LIN {X 0,Y 256.462,Z 255.037,A -85,B 0,C 180,E1 -18622.127,E2 -18622.127} C_VEL
LIN {X 0,Y 256.466,Z 255.038,A -85,B 0,C 180,E1 -18626.861,E2 -18626.861} C_VEL
LIN {X 0,Y 256.7,Z 255.004,A -85,B 0,C 180,E1 -18630.003,E2 -18630.003} C_VEL
LIN {X 0,Y 256.467,Z 255.035,A -85,B 0,C 180,E1 -18633.144,E2 -18633.144} C_VEL
LIN {X 0,Y 256.467,Z 255.036,A -85,B 0,C 180,E1 -18637.878,E2 -18637.878} C_VEL
LIN {X 0,Y 256.243,Z 255.057,A -85,B 0,C 180,E1 -18641.071,E2 -18641.071} C_VEL
LIN {X 0,Y 256.205,Z 255.066,A -85,B 0,C 180,E1 -18645.924,E2 -18645.924} C_VEL
LIN {X 0,Y 256.125,Z 255.068,A -85,B 0,C 180,E1 -18649.227,E2 -18649.227} C_VEL
LIN {X 0,Y 256.028,Z 255.091,A -85,B 0,C 180,E1 -18652.603,E2 -18652.603} C_VEL
LIN {X 0,Y 256.077,Z 255.079,A -85,B 0,C 180,E1 -18656.05,E2 -18656.05} C_VEL
LIN {X 0,Y 256.055,Z 255.069,A -85,B 0,C 180,E1 -18659.61,E2 -18659.61} C_VEL
LIN {X 0,Y 256.039,Z 255.087,A -85,B 0,C 180,E1 -18663.3,E2 -18663.3} C_VEL
LIN {X 0,Y 256.09,Z 255.081,A -85,B 0,C 180,E1 -18667.286,E2 -18667.286} C_VEL
LIN {X 0,Y 256.066,Z 255.085,A -85,B 0,C 180,E1 -18671.204,E2 -18671.204} C_VEL
LIN {X 0,Y 256.081,Z 255.085,A -85,B 0,C 180,E1 -18674.494,E2 -18674.494} C_VEL
LIN {X 0,Y 256.128,Z 255.08,A -85,B 0,C 180,E1 -18678.828,E2 -18678.828} C_VEL
LIN {X 0,Y 256.128,Z 255.078,A -85,B 0,C 180,E1 -18682.883,E2 -18682.883} C_VEL
LIN {X 0,Y 256.062,Z 255.083,A -85,B 0,C 180,E1 -18686.721,E2 -18686.721} C_VEL
LIN {X 0,Y 256.107,Z 255.081,A -85,B 0,C 180,E1 -18691.422,E2 -18691.422} C_VEL
LIN {X 0,Y 256.127,Z 255.076,A -85,B 0,C 180,E1 -18695.708,E2 -18695.708} C_VEL
LIN {X 0,Y 256.115,Z 255.082,A -85,B 0,C 180,E1 -18699.113,E2 -18699.113} C_VEL
LIN {X 0,Y 256.224,Z 255.06,A -85,B 0,C 180,E1 -18704.092,E2 -18704.092} C_VEL
LIN {X 0,Y 256.285,Z 255.059,A -85,B 0,C 180,E1 -18707.339,E2 -18707.339} C_VEL
LIN {X 0,Y 256.435,Z 255.037,A -85,B 0,C 180,E1 -18710.634,E2 -18710.634} C_VEL
LIN {X 0,Y 256.459,Z 255.032,A -85,B 0,C 180,E1 -18713.718,E2 -18713.718} C_VEL
LIN {X 0,Y 256.705,Z 255.007,A -85,B 0,C 180,E1 -18718.442,E2 -18718.442} C_VEL
LIN {X 0,Y 256.708,Z 255.001,A -85,B 0,C 180,E1 -18721.579,E2 -18721.579} C_VEL
LIN {X 0,Y 256.314,Z 255.029,A -85,B 0,C 180,E1 -18724.838,E2 -18724.838} C_VEL
LIN {X 0,Y 255.699,Z 255.11,A -85,B 0,C 180,E1 -18726.152,E2 -18726.152} C_VEL
LIN {X 0,Y 252.868,Z 255.475,A -85,B 0,C 180,E1 -18728.293,E2 -18728.293} C_VEL
LIN {X 0,Y 250.409,Z 255.789,A -85,B 0,C 180,E1 -18730.035,E2 -18730.035} C_VEL
LIN {X 0,Y 249.32,Z 255.926,A -85,B 0,C 180,E1 -18731.387,E2 -18731.387} C_VEL
LIN {X 0,Y 249.215,Z 255.937,A -85,B 0,C 180,E1 -18731.846,E2 -18731.846} C_VEL
LIN {X 0,Y 249.193,Z 255.935,A -85,B 0,C 180,E1 -18736.476,E2 -18736.476} C_VEL
LIN {X 0,Y 249.068,Z 255.955,A -85,B 0,C 180,E1 -18741.53,E2 -18741.53} C_VEL
LIN {X 0,Y 249.107,Z 255.952,A -85,B 0,C 180,E1 -18745.466,E2 -18745.466} C_VEL
LIN {X 0,Y 249.053,Z 255.95,A -85,B 0,C 180,E1 -18748.976,E2 -18748.976} C_VEL
LIN {X 0,Y 249.052,Z 255.96,A -85,B 0,C 180,E1 -18752.433,E2 -18752.433} C_VEL
LIN {X 0,Y 249.038,Z 255.951,A -85,B 0,C 180,E1 -18756.354,E2 -18756.354} C_VEL
LIN {X 0,Y 249.003,Z 255.965,A -85,B 0,C 180,E1 -18760.489,E2 -18760.489} C_VEL
LIN {X 0,Y 248.981,Z 255.971,A -85,B 0,C 180,E1 -18765.113,E2 -18765.113} C_VEL
LIN {X 0,Y 249.001,Z 255.968,A -85,B 0,C 180,E1 -18769.659,E2 -18769.659} C_VEL
LIN {X 0,Y 249.041,Z 255.964,A -85,B 0,C 180,E1 -18773.654,E2 -18773.654} C_VEL
LIN {X 0,Y 249.103,Z 256.071,A -85,B 0,C 180,E1 -18775.646,E2 -18775.646} C_VEL
LIN {X 0,Y 250.915,Z 264.838,A -85,B 0,C 180,E1 -18779.255,E2 -18779.255} C_VEL
LIN {X 0,Y 251.505,Z 267.617,A -85,B 0,C 180,E1 -18780.284,E2 -18780.284} C_VEL
LIN {X 0,Y 258.173,Z 286.572,A -85,B 0,C 180,E1 -18781.623,E2 -18781.623} C_VEL
LIN {X 0,Y 261.815,Z 312.545,A -85,B 0,C 180,E1 -18782.819,E2 -18782.819} C_VEL
LIN {X 0,Y 259.494,Z 375.05,A -85,B 0,C 180,E1 -18784.748,E2 -18784.748} C_VEL
LIN {X 0,Y 258.565,Z 388.595,A -85,B 0,C 180,E1 -18785.456,E2 -18785.456} C_VEL
LIN {X 0,Y 257.311,Z 401.593,A -85,B 0,C 180,E1 -18786.453,E2 -18786.453} C_VEL
LIN {X 0,Y 255.62,Z 414.247,A -85,B 0,C 180,E1 -18787.785,E2 -18787.785} C_VEL
LIN {X 0,Y 253.952,Z 425.589,A -85,B 0,C 180,E1 -18789.336,E2 -18789.336} C_VEL
LIN {X 0,Y 252.459,Z 435.754,A -85,B 0,C 180,E1 -18791.095,E2 -18791.095} C_VEL
LIN {X 0,Y 251.161,Z 444.272,A -85,B 0,C 180,E1 -18792.911,E2 -18792.911} C_VEL
LIN {X 0,Y 249.841,Z 452.028,A -85,B 0,C 180,E1 -18794.915,E2 -18794.915} C_VEL
LIN {X 0,Y 248.545,Z 459.611,A -85,B 0,C 180,E1 -18797.339,E2 -18797.339} C_VEL
LIN {X 0,Y 247.864,Z 464.765,A -85,B 0,C 180,E1 -18799.377,E2 -18799.377} C_VEL
LIN {X 0,Y 247.297,Z 469.736,A -85,B 0,C 180,E1 -18801.828,E2 -18801.828} C_VEL
LIN {X 0,Y 246.944,Z 473.528,A -85,B 0,C 180,E1 -18804.281,E2 -18804.281} C_VEL
LIN {X 0,Y 246.853,Z 476.257,A -85,B 0,C 180,E1 -18806.733,E2 -18806.733} C_VEL
LIN {X 0,Y 246.876,Z 477.532,A -85,B 0,C 180,E1 -18808.366,E2 -18808.366} C_VEL
LIN {X 0,Y 246.908,Z 478.388,A -85,B 0,C 180,E1 -18809.997,E2 -18809.997} C_VEL
LIN {X 0,Y 246.873,Z 478.79,A -85,B 0,C 180,E1 -18811.629,E2 -18811.629} C_VEL
LIN {X 0,Y 246.91,Z 478.408,A -85,B 0,C 180,E1 -18814.896,E2 -18814.896} C_VEL
LIN {X 0,Y 247.108,Z 477.628,A -85,B 0,C 180,E1 -18816.529,E2 -18816.529} C_VEL
LIN {X 0,Y 247.419,Z 476.405,A -85,B 0,C 180,E1 -18818.162,E2 -18818.162} C_VEL
LIN {X 0,Y 248.163,Z 473.816,A -85,B 0,C 180,E1 -18820.605,E2 -18820.605} C_VEL
LIN {X 0,Y 249.262,Z 470.223,A -85,B 0,C 180,E1 -18823.033,E2 -18823.033} C_VEL
LIN {X 0,Y 250.734,Z 465.534,A -85,B 0,C 180,E1 -18825.44,E2 -18825.44} C_VEL
LIN {X 0,Y 253.142,Z 458.477,A -85,B 0,C 180,E1 -18828.197,E2 -18828.197} C_VEL
LIN {X 0,Y 255.47,Z 451.067,A -85,B 0,C 180,E1 -18830.482,E2 -18830.482} C_VEL
LIN {X 0,Y 257.729,Z 443.236,A -85,B 0,C 180,E1 -18832.44,E2 -18832.44} C_VEL
LIN {X 0,Y 260.587,Z 432.866,A -85,B 0,C 180,E1 -18834.495,E2 -18834.495} C_VEL
LIN {X 0,Y 263.36,Z 422.361,A -85,B 0,C 180,E1 -18836.121,E2 -18836.121} C_VEL
LIN {X 0,Y 265.495,Z 412.353,A -85,B 0,C 180,E1 -18837.38,E2 -18837.38} C_VEL
LIN {X 0,Y 267.92,Z 399.574,A -85,B 0,C 180,E1 -18838.599,E2 -18838.599} C_VEL
LIN {X 0,Y 269.848,Z 386.608,A -85,B 0,C 180,E1 -18839.495,E2 -18839.495} C_VEL
LIN {X 0,Y 271.208,Z 373.712,A -85,B 0,C 180,E1 -18840.096,E2 -18840.096} C_VEL
LIN {X 0,Y 274.368,Z 315.731,A -85,B 0,C 180,E1 -18841.897,E2 -18841.897} C_VEL
LIN {X 0,Y 272.677,Z 304.843,A -85,B 0,C 180,E1 -18842.649,E2 -18842.649} C_VEL
LIN {X 0,Y 268.046,Z 294.247,A -85,B 0,C 180,E1 -18843.981,E2 -18843.981} C_VEL
LIN {X 0,Y 262.592,Z 283.414,A -85,B 0,C 180,E1 -18845.624,E2 -18845.624} C_VEL
LIN {X 0,Y 257.789,Z 275.094,A -85,B 0,C 180,E1 -18847.131,E2 -18847.131} C_VEL
LIN {X 0,Y 254.919,Z 270.398,A -85,B 0,C 180,E1 -18848.092,E2 -18848.092} C_VEL
LIN {X 0,Y 252.035,Z 265.64,A -85,B 0,C 180,E1 -18849.18,E2 -18849.18} C_VEL
LIN {X 0,Y 249.945,Z 259.149,A -85,B 0,C 180,E1 -18853.012,E2 -18853.012} C_VEL
LIN {X 0,Y 249.001,Z 256,A -85,B 0,C 180,E1 -18855.252,E2 -18855.252} C_VEL
LIN {X 0,Y 248.992,Z 255.969,A -85,B 0,C 180,E1 -18859.644,E2 -18859.644} C_VEL
LIN {X 0,Y 249.019,Z 255.958,A -85,B 0,C 180,E1 -18863.643,E2 -18863.643} C_VEL
LIN {X 0,Y 249.037,Z 255.96,A -85,B 0,C 180,E1 -18867.84,E2 -18867.84} C_VEL
LIN {X 0,Y 249.043,Z 255.96,A -85,B 0,C 180,E1 -18871.322,E2 -18871.322} C_VEL
LIN {X 0,Y 249.103,Z 255.952,A -85,B 0,C 180,E1 -18874.954,E2 -18874.954} C_VEL
LIN {X 0,Y 249.053,Z 255.96,A -85,B 0,C 180,E1 -18878.617,E2 -18878.617} C_VEL
LIN {X 0,Y 249.155,Z 255.943,A -85,B 0,C 180,E1 -18883.606,E2 -18883.606} C_VEL
LIN {X 0,Y 249.212,Z 255.935,A -85,B 0,C 180,E1 -18888.605,E2 -18888.605} C_VEL
LIN {X 0,Y 249.406,Z 255.912,A -85,B 0,C 180,E1 -18891.89,E2 -18891.89} C_VEL
LIN {X 0,Y 249.255,Z 255.932,A -85,B 0,C 180,E1 -18895.137,E2 -18895.137} C_VEL
LIN {X 0,Y 249.648,Z 255.887,A -85,B 0,C 180,E1 -18898.376,E2 -18898.376} C_VEL
LIN {X 0,Y 249.657,Z 255.886,A -85,B 0,C 180,E1 -18901.602,E2 -18901.602} C_VEL
LIN {X 0,Y 249.451,Z 256.029,A -85,B 0,C 180,E1 -18903.219,E2 -18903.219} C_VEL
LIN {X 0,Y 251.162,Z 261.37,A -85,B 0,C 180,E1 -18906.617,E2 -18906.617} C_VEL
LIN {X 0,Y 254.131,Z 265.956,A -85,B 0,C 180,E1 -18907.737,E2 -18907.737} C_VEL
LIN {X 0,Y 258.847,Z 273.575,A -85,B 0,C 180,E1 -18909.315,E2 -18909.315} C_VEL
LIN {X 0,Y 265.164,Z 284.458,A -85,B 0,C 180,E1 -18911.246,E2 -18911.246} C_VEL
LIN {X 0,Y 270.999,Z 296.328,A -85,B 0,C 180,E1 -18912.943,E2 -18912.943} C_VEL
LIN {X 0,Y 274.837,Z 305.474,A -85,B 0,C 180,E1 -18914.031,E2 -18914.031} C_VEL
LIN {X 0,Y 271.212,Z 369.796,A -85,B 0,C 180,E1 -18916.039,E2 -18916.039} C_VEL
LIN {X 0,Y 269.677,Z 383.672,A -85,B 0,C 180,E1 -18916.745,E2 -18916.745} C_VEL
LIN {X 0,Y 268.02,Z 395.502,A -85,B 0,C 180,E1 -18917.638,E2 -18917.638} C_VEL
LIN {X 0,Y 265.705,Z 407.921,A -85,B 0,C 180,E1 -18918.894,E2 -18918.894} C_VEL
LIN {X 0,Y 263.365,Z 418.563,A -85,B 0,C 180,E1 -18920.286,E2 -18920.286} C_VEL
LIN {X 0,Y 260.75,Z 428.824,A -85,B 0,C 180,E1 -18921.968,E2 -18921.968} C_VEL
LIN {X 0,Y 258.22,Z 437.668,A -85,B 0,C 180,E1 -18923.782,E2 -18923.782} C_VEL
LIN {X 0,Y 255.435,Z 446.676,A -85,B 0,C 180,E1 -18926.105,E2 -18926.105} C_VEL
LIN {X 0,Y 252.942,Z 454.285,A -85,B 0,C 180,E1 -18928.599,E2 -18928.599} C_VEL
LIN {X 0,Y 250.854,Z 460.406,A -85,B 0,C 180,E1 -18931.204,E2 -18931.204} C_VEL
LIN {X 0,Y 249.511,Z 464.384,A -85,B 0,C 180,E1 -18933.369,E2 -18933.369} C_VEL
LIN {X 0,Y 248.057,Z 468.539,A -85,B 0,C 180,E1 -18936.495,E2 -18936.495} C_VEL
LIN {X 0,Y 247.091,Z 471.202,A -85,B 0,C 180,E1 -18939.834,E2 -18939.834} C_VEL
LIN {X 0,Y 246.59,Z 472.14,A -85,B 0,C 180,E1 -18943.14,E2 -18943.14} C_VEL
LIN {X 0,Y 246.467,Z 471.807,A -85,B 0,C 180,E1 -18945.45,E2 -18945.45} C_VEL
LIN {X 0,Y 246.455,Z 470.618,A -85,B 0,C 180,E1 -18947.832,E2 -18947.832} C_VEL
LIN {X 0,Y 246.642,Z 468.47,A -85,B 0,C 180,E1 -18950.275,E2 -18950.275} C_VEL
LIN {X 0,Y 247.058,Z 465.231,A -85,B 0,C 180,E1 -18952.775,E2 -18952.775} C_VEL
LIN {X 0,Y 247.691,Z 460.527,A -85,B 0,C 180,E1 -18955.429,E2 -18955.429} C_VEL
LIN {X 0,Y 248.603,Z 454.629,A -85,B 0,C 180,E1 -18957.979,E2 -18957.979} C_VEL
LIN {X 0,Y 249.514,Z 448.37,A -85,B 0,C 180,E1 -18960.142,E2 -18960.142} C_VEL
LIN {X 0,Y 250.916,Z 440.001,A -85,B 0,C 180,E1 -18962.478,E2 -18962.478} C_VEL
LIN {X 0,Y 252.491,Z 430.143,A -85,B 0,C 180,E1 -18964.665,E2 -18964.665} C_VEL
LIN {X 0,Y 254.061,Z 420.365,A -85,B 0,C 180,E1 -18966.41,E2 -18966.41} C_VEL
LIN {X 0,Y 255.514,Z 410.22,A -85,B 0,C 180,E1 -18967.875,E2 -18967.875} C_VEL
LIN {X 0,Y 257.062,Z 397.642,A -85,B 0,C 180,E1 -18969.289,E2 -18969.289} C_VEL
LIN {X 0,Y 258.251,Z 385.45,A -85,B 0,C 180,E1 -18970.323,E2 -18970.323} C_VEL
LIN {X 0,Y 259.236,Z 373.09,A -85,B 0,C 180,E1 -18971.065,E2 -18971.065} C_VEL
LIN {X 0,Y 260.034,Z 356.998,A -85,B 0,C 180,E1 -18971.647,E2 -18971.647} C_VEL
LIN {X 0,Y 262.026,Z 299.434,A -85,B 0,C 180,E1 -18973.409,E2 -18973.409} C_VEL
LIN {X 0,Y 260.034,Z 288.531,A -85,B 0,C 180,E1 -18973.952,E2 -18973.952} C_VEL
LIN {X 0,Y 250.328,Z 261.517,A -85,B 0,C 180,E1 -18975.834,E2 -18975.834} C_VEL
LIN {X 0,Y 250.056,Z 260.316,A -85,B 0,C 180,E1 -18976.182,E2 -18976.182} C_VEL
LIN {X 0,Y 249.212,Z 256.009,A -85,B 0,C 180,E1 -18978.102,E2 -18978.102} C_VEL
LIN {X 0,Y 249.4,Z 255.917,A -85,B 0,C 180,E1 -18981.903,E2 -18981.903} C_VEL
LIN {X 0,Y 249.401,Z 255.917,A -85,B 0,C 180,E1 -18986.772,E2 -18986.772} C_VEL
LIN {X 0,Y 249.663,Z 255.88,A -85,B 0,C 180,E1 -18990.003,E2 -18990.003} C_VEL
LIN {X 0,Y 249.401,Z 255.914,A -85,B 0,C 180,E1 -18993.234,E2 -18993.234} C_VEL
LIN {X 0,Y 249.408,Z 255.915,A -85,B 0,C 180,E1 -18998.102,E2 -18998.102} C_VEL
LIN {X 0,Y 249.183,Z 255.938,A -85,B 0,C 180,E1 -19001.389,E2 -19001.389} C_VEL
LIN {X 0,Y 249.139,Z 255.944,A -85,B 0,C 180,E1 -19006.492,E2 -19006.492} C_VEL
LIN {X 0,Y 249.03,Z 255.962,A -85,B 0,C 180,E1 -19011.526,E2 -19011.526} C_VEL
LIN {X 0,Y 249.065,Z 255.958,A -85,B 0,C 180,E1 -19015.483,E2 -19015.483} C_VEL
LIN {X 0,Y 249.024,Z 255.941,A -85,B 0,C 180,E1 -19018.998,E2 -19018.998} C_VEL
LIN {X 0,Y 248.99,Z 255.967,A -85,B 0,C 180,E1 -19022.435,E2 -19022.435} C_VEL
LIN {X 0,Y 249.027,Z 255.965,A -85,B 0,C 180,E1 -19026.349,E2 -19026.349} C_VEL
LIN {X 0,Y 249.039,Z 255.962,A -85,B 0,C 180,E1 -19030.475,E2 -19030.475} C_VEL
LIN {X 0,Y 249.027,Z 255.961,A -85,B 0,C 180,E1 -19034.877,E2 -19034.877} C_VEL
LIN {X 0,Y 249.065,Z 255.953,A -85,B 0,C 180,E1 -19037.391,E2 -19037.391} C_VEL
LIN {X 0,Y 249.044,Z 255.96,A -85,B 0,C 180,E1 -19041.639,E2 -19041.639} C_VEL
LIN {X 0,Y 249.037,Z 255.955,A -85,B 0,C 180,E1 -19045.654,E2 -19045.654} C_VEL
LIN {X 0,Y 249.027,Z 255.964,A -85,B 0,C 180,E1 -19049.484,E2 -19049.484} C_VEL
LIN {X 0,Y 249.051,Z 255.956,A -85,B 0,C 180,E1 -19053.174,E2 -19053.174} C_VEL
LIN {X 0,Y 249.044,Z 255.957,A -85,B 0,C 180,E1 -19056.742,E2 -19056.742} C_VEL
LIN {X 0,Y 249.049,Z 255.959,A -85,B 0,C 180,E1 -19060.219,E2 -19060.219} C_VEL
LIN {X 0,Y 249.152,Z 255.941,A -85,B 0,C 180,E1 -19063.628,E2 -19063.628} C_VEL
LIN {X 0,Y 249.209,Z 255.938,A -85,B 0,C 180,E1 -19066.973,E2 -19066.973} C_VEL
LIN {X 0,Y 249.384,Z 255.916,A -85,B 0,C 180,E1 -19070.534,E2 -19070.534} C_VEL
LIN {X 0,Y 249.43,Z 255.906,A -85,B 0,C 180,E1 -19073.54,E2 -19073.54} C_VEL
LIN {X 0,Y 249.666,Z 255.884,A -85,B 0,C 180,E1 -19078.398,E2 -19078.398} C_VEL
LIN {X 0,Y 249.669,Z 255.878,A -85,B 0,C 180,E1 -19081.624,E2 -19081.624} C_VEL
LIN {X 0,Y 249.438,Z 255.89,A -85,B 0,C 180,E1 -19086.481,E2 -19086.481} C_VEL
LIN {X 0,Y 249.35,Z 255.918,A -85,B 0,C 180,E1 -19089.746,E2 -19089.746} C_VEL
LIN {X 0,Y 249.215,Z 255.937,A -85,B 0,C 180,E1 -19091.846,E2 -19091.846} C_VEL
LIN {X 0,Y 248.503,Z 256.029,A -85,B 0,C 180,E1 -19093.195,E2 -19093.195} C_VEL
LIN {X 0,Y 245.629,Z 256.381,A -85,B 0,C 180,E1 -19095.394,E2 -19095.394} C_VEL
LIN {X 0,Y 243.193,Z 256.677,A -85,B 0,C 180,E1 -19097.185,E2 -19097.185} C_VEL
LIN {X 0,Y 242.119,Z 256.806,A -85,B 0,C 180,E1 -19098.574,E2 -19098.574} C_VEL
LIN {X 0,Y 242.015,Z 256.818,A -85,B 0,C 180,E1 -19099.045,E2 -19099.045} C_VEL
LIN {X 0,Y 242.01,Z 256.834,A -85,B 0,C 180,E1 -19102.19,E2 -19102.19} C_VEL
LIN {X 0,Y 242.058,Z 256.829,A -85,B 0,C 180,E1 -19105.828,E2 -19105.828} C_VEL
LIN {X 0,Y 241.99,Z 256.831,A -85,B 0,C 180,E1 -19109.596,E2 -19109.596} C_VEL
LIN {X 0,Y 242.006,Z 256.839,A -85,B 0,C 180,E1 -19113.499,E2 -19113.499} C_VEL
LIN {X 0,Y 242.011,Z 256.833,A -85,B 0,C 180,E1 -19117.589,E2 -19117.589} C_VEL
LIN {X 0,Y 241.91,Z 256.844,A -85,B 0,C 180,E1 -19121.939,E2 -19121.939} C_VEL
LIN {X 0,Y 241.913,Z 256.848,A -85,B 0,C 180,E1 -19125.791,E2 -19125.791} C_VEL
LIN {X 0,Y 241.958,Z 256.846,A -85,B 0,C 180,E1 -19130.278,E2 -19130.278} C_VEL
LIN {X 0,Y 242.005,Z 256.841,A -85,B 0,C 180,E1 -19134.489,E2 -19134.489} C_VEL
LIN {X 0,Y 242.091,Z 257.09,A -85,B 0,C 180,E1 -19135.266,E2 -19135.266} C_VEL
LIN {X 0,Y 244.176,Z 267.14,A -85,B 0,C 180,E1 -19139.444,E2 -19139.444} C_VEL
LIN {X 0,Y 244.512,Z 268.458,A -85,B 0,C 180,E1 -19139.658,E2 -19139.658} C_VEL
LIN {X 0,Y 251.727,Z 288.53,A -85,B 0,C 180,E1 -19141.095,E2 -19141.095} C_VEL
LIN {X 0,Y 255.157,Z 313.421,A -85,B 0,C 180,E1 -19142.281,E2 -19142.281} C_VEL
LIN {X 0,Y 252.768,Z 375.344,A -85,B 0,C 180,E1 -19144.248,E2 -19144.248} C_VEL
LIN {X 0,Y 251.816,Z 388.749,A -85,B 0,C 180,E1 -19144.973,E2 -19144.973} C_VEL
LIN {X 0,Y 250.533,Z 401.676,A -85,B 0,C 180,E1 -19145.996,E2 -19145.996} C_VEL
LIN {X 0,Y 248.779,Z 414.28,A -85,B 0,C 180,E1 -19147.359,E2 -19147.359} C_VEL
LIN {X 0,Y 247.07,Z 425.601,A -85,B 0,C 180,E1 -19148.951,E2 -19148.951} C_VEL
LIN {X 0,Y 245.604,Z 435.311,A -85,B 0,C 180,E1 -19150.67,E2 -19150.67} C_VEL
LIN {X 0,Y 244.022,Z 445.078,A -85,B 0,C 180,E1 -19152.827,E2 -19152.827} C_VEL
LIN {X 0,Y 242.476,Z 454.073,A -85,B 0,C 180,E1 -19155.306,E2 -19155.306} C_VEL
LIN {X 0,Y 241.272,Z 461.233,A -85,B 0,C 180,E1 -19157.805,E2 -19157.805} C_VEL
LIN {X 0,Y 240.414,Z 467.764,A -85,B 0,C 180,E1 -19160.745,E2 -19160.745} C_VEL
LIN {X 0,Y 239.986,Z 472.022,A -85,B 0,C 180,E1 -19163.27,E2 -19163.27} C_VEL
LIN {X 0,Y 239.798,Z 474.602,A -85,B 0,C 180,E1 -19165.271,E2 -19165.271} C_VEL
LIN {X 0,Y 239.79,Z 477.299,A -85,B 0,C 180,E1 -19168.318,E2 -19168.318} C_VEL
LIN {X 0,Y 239.821,Z 478.201,A -85,B 0,C 180,E1 -19169.997,E2 -19169.997} C_VEL
LIN {X 0,Y 239.787,Z 478.67,A -85,B 0,C 180,E1 -19171.677,E2 -19171.677} C_VEL
LIN {X 0,Y 239.83,Z 478.367,A -85,B 0,C 180,E1 -19175.041,E2 -19175.041} C_VEL
LIN {X 0,Y 240.058,Z 477.633,A -85,B 0,C 180,E1 -19176.722,E2 -19176.722} C_VEL
LIN {X 0,Y 240.394,Z 476.482,A -85,B 0,C 180,E1 -19178.402,E2 -19178.402} C_VEL
LIN {X 0,Y 241.174,Z 473.968,A -85,B 0,C 180,E1 -19180.916,E2 -19180.916} C_VEL
LIN {X 0,Y 242.34,Z 470.45,A -85,B 0,C 180,E1 -19183.412,E2 -19183.412} C_VEL
LIN {X 0,Y 243.892,Z 465.875,A -85,B 0,C 180,E1 -19185.884,E2 -19185.884} C_VEL
LIN {X 0,Y 246.434,Z 458.967,A -85,B 0,C 180,E1 -19188.71,E2 -19188.71} C_VEL
LIN {X 0,Y 248.797,Z 451.904,A -85,B 0,C 180,E1 -19190.987,E2 -19190.987} C_VEL
LIN {X 0,Y 251.242,Z 443.99,A -85,B 0,C 180,E1 -19193.052,E2 -19193.052} C_VEL
LIN {X 0,Y 253.996,Z 434.893,A -85,B 0,C 180,E1 -19194.955,E2 -19194.955} C_VEL
LIN {X 0,Y 256.777,Z 424.851,A -85,B 0,C 180,E1 -19196.624,E2 -19196.624} C_VEL
LIN {X 0,Y 259.313,Z 413.919,A -85,B 0,C 180,E1 -19198.09,E2 -19198.09} C_VEL
LIN {X 0,Y 261.868,Z 401.783,A -85,B 0,C 180,E1 -19199.323,E2 -19199.323} C_VEL
LIN {X 0,Y 263.693,Z 390.48,A -85,B 0,C 180,E1 -19200.199,E2 -19200.199} C_VEL
LIN {X 0,Y 265.324,Z 377.226,A -85,B 0,C 180,E1 -19200.906,E2 -19200.906} C_VEL
LIN {X 0,Y 266.636,Z 357.045,A -85,B 0,C 180,E1 -19201.591,E2 -19201.591} C_VEL
LIN {X 0,Y 268.965,Z 317.109,A -85,B 0,C 180,E1 -19202.827,E2 -19202.827} C_VEL
LIN {X 0,Y 267.623,Z 308.149,A -85,B 0,C 180,E1 -19203.465,E2 -19203.465} C_VEL
LIN {X 0,Y 262.848,Z 296.901,A -85,B 0,C 180,E1 -19204.951,E2 -19204.951} C_VEL
LIN {X 0,Y 256.9,Z 285.254,A -85,B 0,C 180,E1 -19206.846,E2 -19206.846} C_VEL
LIN {X 0,Y 251.429,Z 275.929,A -85,B 0,C 180,E1 -19208.724,E2 -19208.724} C_VEL
LIN {X 0,Y 247.851,Z 270.43,A -85,B 0,C 180,E1 -19210.027,E2 -19210.027} C_VEL
LIN {X 0,Y 245.42,Z 266.863,A -85,B 0,C 180,E1 -19210.969,E2 -19210.969} C_VEL
LIN {X 0,Y 244.666,Z 265.35,A -85,B 0,C 180,E1 -19211.391,E2 -19211.391} C_VEL
LIN {X 0,Y 243.132,Z 260.625,A -85,B 0,C 180,E1 -19214.467,E2 -19214.467} C_VEL
LIN {X 0,Y 241.97,Z 256.888,A -85,B 0,C 180,E1 -19217.377,E2 -19217.377} C_VEL
LIN {X 0,Y 241.992,Z 256.842,A -85,B 0,C 180,E1 -19222.408,E2 -19222.408} C_VEL
LIN {X 0,Y 241.986,Z 256.834,A -85,B 0,C 180,E1 -19226.498,E2 -19226.498} C_VEL
LIN {X 0,Y 241.977,Z 256.835,A -85,B 0,C 180,E1 -19230.605,E2 -19230.605} C_VEL
LIN {X 0,Y 242.036,Z 256.826,A -85,B 0,C 180,E1 -19234.169,E2 -19234.169} C_VEL
LIN {X 0,Y 241.992,Z 256.836,A -85,B 0,C 180,E1 -19238.324,E2 -19238.324} C_VEL
LIN {X 0,Y 242.103,Z 256.823,A -85,B 0,C 180,E1 -19243.314,E2 -19243.314} C_VEL
LIN {X 0,Y 242.146,Z 256.813,A -85,B 0,C 180,E1 -19248.267,E2 -19248.267} C_VEL
LIN {X 0,Y 242.36,Z 256.788,A -85,B 0,C 180,E1 -19251.653,E2 -19251.653} C_VEL
LIN {X 0,Y 242.388,Z 256.789,A -85,B 0,C 180,E1 -19253.329,E2 -19253.329} C_VEL
LIN {X 0,Y 242.608,Z 256.763,A -85,B 0,C 180,E1 -19258.329,E2 -19258.329} C_VEL
LIN {X 0,Y 242.63,Z 256.926,A -85,B 0,C 180,E1 -19261.234,E2 -19261.234} C_VEL
LIN {X 0,Y 243.86,Z 261.641,A -85,B 0,C 180,E1 -19264.431,E2 -19264.431} C_VEL
LIN {X 0,Y 246.894,Z 266.121,A -85,B 0,C 180,E1 -19265.706,E2 -19265.706} C_VEL
LIN {X 0,Y 248.442,Z 268.242,A -85,B 0,C 180,E1 -19266.29,E2 -19266.29} C_VEL
LIN {X 0,Y 251.808,Z 273.304,A -85,B 0,C 180,E1 -19267.506,E2 -19267.506} C_VEL
LIN {X 0,Y 257.832,Z 283.574,A -85,B 0,C 180,E1 -19269.563,E2 -19269.563} C_VEL
LIN {X 0,Y 262.904,Z 293.011,A -85,B 0,C 180,E1 -19271.148,E2 -19271.148} C_VEL
LIN {X 0,Y 267.924,Z 304.094,A -85,B 0,C 180,E1 -19272.686,E2 -19272.686} C_VEL
LIN {X 0,Y 269.444,Z 307.892,A -85,B 0,C 180,E1 -19273.137,E2 -19273.137} C_VEL
LIN {X 0,Y 265.705,Z 369.852,A -85,B 0,C 180,E1 -19275.088,E2 -19275.088} C_VEL
LIN {X 0,Y 264.07,Z 383.999,A -85,B 0,C 180,E1 -19275.821,E2 -19275.821} C_VEL
LIN {X 0,Y 262.303,Z 395.777,A -85,B 0,C 180,E1 -19276.729,E2 -19276.729} C_VEL
LIN {X 0,Y 259.853,Z 408.216,A -85,B 0,C 180,E1 -19278.017,E2 -19278.017} C_VEL
LIN {X 0,Y 257.196,Z 419.554,A -85,B 0,C 180,E1 -19279.544,E2 -19279.544} C_VEL
LIN {X 0,Y 254.483,Z 429.525,A -85,B 0,C 180,E1 -19281.239,E2 -19281.239} C_VEL
LIN {X 0,Y 251.344,Z 439.839,A -85,B 0,C 180,E1 -19283.467,E2 -19283.467} C_VEL
LIN {X 0,Y 248.663,Z 448,A -85,B 0,C 180,E1 -19285.702,E2 -19285.702} C_VEL
LIN {X 0,Y 245.892,Z 455.746,A -85,B 0,C 180,E1 -19288.433,E2 -19288.433} C_VEL
LIN {X 0,Y 243.683,Z 461.858,A -85,B 0,C 180,E1 -19291.259,E2 -19291.259} C_VEL
LIN {X 0,Y 241.884,Z 466.763,A -85,B 0,C 180,E1 -19294.402,E2 -19294.402} C_VEL
LIN {X 0,Y 240.488,Z 470.302,A -85,B 0,C 180,E1 -19297.841,E2 -19297.841} C_VEL
LIN {X 0,Y 239.884,Z 471.746,A -85,B 0,C 180,E1 -19300.388,E2 -19300.388} C_VEL
LIN {X 0,Y 239.529,Z 472.242,A -85,B 0,C 180,E1 -19302.823,E2 -19302.823} C_VEL
LIN {X 0,Y 239.385,Z 471.916,A -85,B 0,C 180,E1 -19305.207,E2 -19305.207} C_VEL
LIN {X 0,Y 239.346,Z 470.831,A -85,B 0,C 180,E1 -19307.523,E2 -19307.523} C_VEL
LIN {X 0,Y 239.491,Z 469.004,A -85,B 0,C 180,E1 -19309.794,E2 -19309.794} C_VEL
LIN {X 0,Y 239.881,Z 466.085,A -85,B 0,C 180,E1 -19312.26,E2 -19312.26} C_VEL
LIN {X 0,Y 240.467,Z 461.839,A -85,B 0,C 180,E1 -19314.894,E2 -19314.894} C_VEL
LIN {X 0,Y 241.318,Z 456.064,A -85,B 0,C 180,E1 -19317.6,E2 -19317.6} C_VEL
LIN {X 0,Y 242.49,Z 448.458,A -85,B 0,C 180,E1 -19320.369,E2 -19320.369} C_VEL
LIN {X 0,Y 243.782,Z 440.994,A -85,B 0,C 180,E1 -19322.535,E2 -19322.535} C_VEL
LIN {X 0,Y 245.197,Z 432.544,A -85,B 0,C 180,E1 -19324.54,E2 -19324.54} C_VEL
LIN {X 0,Y 246.904,Z 422.154,A -85,B 0,C 180,E1 -19326.519,E2 -19326.519} C_VEL
LIN {X 0,Y 248.577,Z 410.948,A -85,B 0,C 180,E1 -19328.221,E2 -19328.221} C_VEL
LIN {X 0,Y 250.165,Z 398.722,A -85,B 0,C 180,E1 -19329.659,E2 -19329.659} C_VEL
LIN {X 0,Y 251.463,Z 386.124,A -85,B 0,C 180,E1 -19330.772,E2 -19330.772} C_VEL
LIN {X 0,Y 252.518,Z 373.317,A -85,B 0,C 180,E1 -19331.571,E2 -19331.571} C_VEL
LIN {X 0,Y 253.314,Z 357.756,A -85,B 0,C 180,E1 -19332.154,E2 -19332.154} C_VEL
LIN {X 0,Y 255.393,Z 300.126,A -85,B 0,C 180,E1 -19333.964,E2 -19333.964} C_VEL
LIN {X 0,Y 253.57,Z 290.539,A -85,B 0,C 180,E1 -19334.463,E2 -19334.463} C_VEL
LIN {X 0,Y 244.047,Z 264.077,A -85,B 0,C 180,E1 -19336.339,E2 -19336.339} C_VEL
LIN {X 0,Y 243.023,Z 261.254,A -85,B 0,C 180,E1 -19336.626,E2 -19336.626} C_VEL
LIN {X 0,Y 242.173,Z 256.889,A -85,B 0,C 180,E1 -19338.547,E2 -19338.547} C_VEL
LIN {X 0,Y 242.349,Z 256.796,A -85,B 0,C 180,E1 -19341.666,E2 -19341.666} C_VEL
LIN {X 0,Y 242.202,Z 256.812,A -85,B 0,C 180,E1 -19345.009,E2 -19345.009} C_VEL
LIN {X 0,Y 242.581,Z 256.768,A -85,B 0,C 180,E1 -19348.343,E2 -19348.343} C_VEL
LIN {X 0,Y 242.581,Z 256.767,A -85,B 0,C 180,E1 -19351.663,E2 -19351.663} C_VEL
LIN {X 0,Y 242.367,Z 256.793,A -85,B 0,C 180,E1 -19356.663,E2 -19356.663} C_VEL
LIN {X 0,Y 242.252,Z 256.797,A -85,B 0,C 180,E1 -19360.027,E2 -19360.027} C_VEL
LIN {X 0,Y 242.083,Z 256.83,A -85,B 0,C 180,E1 -19365.149,E2 -19365.149} C_VEL
LIN {X 0,Y 242.009,Z 256.823,A -85,B 0,C 180,E1 -19368.632,E2 -19368.632} C_VEL
LIN {X 0,Y 241.953,Z 256.846,A -85,B 0,C 180,E1 -19372.189,E2 -19372.189} C_VEL
LIN {X 0,Y 242.017,Z 256.831,A -85,B 0,C 180,E1 -19375.847,E2 -19375.847} C_VEL
LIN {X 0,Y 241.959,Z 256.822,A -85,B 0,C 180,E1 -19379.593,E2 -19379.593} C_VEL
LIN {X 0,Y 241.946,Z 256.843,A -85,B 0,C 180,E1 -19383.501,E2 -19383.501} C_VEL
LIN {X 0,Y 241.966,Z 256.841,A -85,B 0,C 180,E1 -19387.589,E2 -19387.589} C_VEL
LIN {X 0,Y 241.957,Z 256.844,A -85,B 0,C 180,E1 -19391.921,E2 -19391.921} C_VEL
LIN {X 0,Y 241.99,Z 256.835,A -85,B 0,C 180,E1 -19396.56,E2 -19396.56} C_VEL
LIN {X 0,Y 241.995,Z 256.839,A -85,B 0,C 180,E1 -19400.306,E2 -19400.306} C_VEL
LIN {X 0,Y 242.012,Z 256.833,A -85,B 0,C 180,E1 -19404.51,E2 -19404.51} C_VEL
LIN {X 0,Y 241.953,Z 256.843,A -85,B 0,C 180,E1 -19408.492,E2 -19408.492} C_VEL
LIN {X 0,Y 241.982,Z 256.838,A -85,B 0,C 180,E1 -19412.324,E2 -19412.324} C_VEL
LIN {X 0,Y 242.025,Z 256.831,A -85,B 0,C 180,E1 -19416.026,E2 -19416.026} C_VEL
LIN {X 0,Y 241.984,Z 256.842,A -85,B 0,C 180,E1 -19419.616,E2 -19419.616} C_VEL
LIN {X 0,Y 242.107,Z 256.82,A -85,B 0,C 180,E1 -19423.33,E2 -19423.33} C_VEL
LIN {X 0,Y 242.176,Z 256.816,A -85,B 0,C 180,E1 -19428.291,E2 -19428.291} C_VEL
LIN {X 0,Y 242.373,Z 256.789,A -85,B 0,C 180,E1 -19431.675,E2 -19431.675} C_VEL
LIN {X 0,Y 242.4,Z 256.78,A -85,B 0,C 180,E1 -19433.352,E2 -19433.352} C_VEL
LIN {X 0,Y 242.626,Z 256.761,A -85,B 0,C 180,E1 -19438.351,E2 -19438.351} C_VEL
LIN {X 0,Y 242.628,Z 256.754,A -85,B 0,C 180,E1 -19441.671,E2 -19441.671} C_VEL
LIN {X 0,Y 242.409,Z 256.766,A -85,B 0,C 180,E1 -19446.67,E2 -19446.67} C_VEL
LIN {X 0,Y 242.278,Z 256.8,A -85,B 0,C 180,E1 -19450.034,E2 -19450.034} C_VEL
LIN {X 0,Y 242.141,Z 256.816,A -85,B 0,C 180,E1 -19455.153,E2 -19455.153} C_VEL
LIN {X 0,Y 242.015,Z 256.818,A -85,B 0,C 180,E1 -19459.045,E2 -19459.045} C_VEL
LIN {X 0,Y 241.317,Z 256.913,A -85,B 0,C 180,E1 -19460.433,E2 -19460.433} C_VEL
LIN {X 0,Y 238.508,Z 257.273,A -85,B 0,C 180,E1 -19462.699,E2 -19462.699} C_VEL
LIN {X 0,Y 235.319,Z 257.671,A -85,B 0,C 180,E1 -19465.492,E2 -19465.492} C_VEL
LIN {X 0,Y 234.977,Z 257.71,A -85,B 0,C 180,E1 -19466.458,E2 -19466.458} C_VEL
LIN {X 0,Y 234.922,Z 257.714,A -85,B 0,C 180,E1 -19470.58,E2 -19470.58} C_VEL
LIN {X 0,Y 234.95,Z 257.716,A -85,B 0,C 180,E1 -19474.646,E2 -19474.646} C_VEL
LIN {X 0,Y 234.941,Z 257.718,A -85,B 0,C 180,E1 -19478.94,E2 -19478.94} C_VEL
LIN {X 0,Y 234.879,Z 257.728,A -85,B 0,C 180,E1 -19484.097,E2 -19484.097} C_VEL
LIN {X 0,Y 234.863,Z 257.729,A -85,B 0,C 180,E1 -19488.825,E2 -19488.825} C_VEL
LIN {X 0,Y 234.95,Z 257.719,A -85,B 0,C 180,E1 -19491.082,E2 -19491.082} C_VEL
LIN {X 0,Y 235.024,Z 257.917,A -85,B 0,C 180,E1 -19494.744,E2 -19494.744} C_VEL
LIN {X 0,Y 236.952,Z 267.222,A -85,B 0,C 180,E1 -19498.742,E2 -19498.742} C_VEL
LIN {X 0,Y 238.193,Z 270.731,A -85,B 0,C 180,E1 -19499.114,E2 -19499.114} C_VEL
LIN {X 0,Y 245.394,Z 290.901,A -85,B 0,C 180,E1 -19500.589,E2 -19500.589} C_VEL
LIN {X 0,Y 248.5,Z 314.507,A -85,B 0,C 180,E1 -19501.726,E2 -19501.726} C_VEL
LIN {X 0,Y 246.062,Z 375.357,A -85,B 0,C 180,E1 -19503.72,E2 -19503.72} C_VEL
LIN {X 0,Y 244.995,Z 389.426,A -85,B 0,C 180,E1 -19504.511,E2 -19504.511} C_VEL
LIN {X 0,Y 243.766,Z 401.601,A -85,B 0,C 180,E1 -19505.513,E2 -19505.513} C_VEL
LIN {X 0,Y 241.952,Z 414.183,A -85,B 0,C 180,E1 -19506.91,E2 -19506.91} C_VEL
LIN {X 0,Y 240.201,Z 425.499,A -85,B 0,C 180,E1 -19508.544,E2 -19508.544} C_VEL
LIN {X 0,Y 238.581,Z 435.74,A -85,B 0,C 180,E1 -19510.421,E2 -19510.421} C_VEL
LIN {X 0,Y 236.878,Z 445.802,A -85,B 0,C 180,E1 -19512.738,E2 -19512.738} C_VEL
LIN {X 0,Y 235.558,Z 453.275,A -85,B 0,C 180,E1 -19514.864,E2 -19514.864} C_VEL
LIN {X 0,Y 234.293,Z 460.604,A -85,B 0,C 180,E1 -19517.436,E2 -19517.436} C_VEL
LIN {X 0,Y 233.606,Z 465.538,A -85,B 0,C 180,E1 -19519.598,E2 -19519.598} C_VEL
LIN {X 0,Y 233.035,Z 470.299,A -85,B 0,C 180,E1 -19522.197,E2 -19522.197} C_VEL
LIN {X 0,Y 232.707,Z 474.549,A -85,B 0,C 180,E1 -19525.389,E2 -19525.389} C_VEL
LIN {X 0,Y 232.688,Z 477.056,A -85,B 0,C 180,E1 -19528.266,E2 -19528.266} C_VEL
LIN {X 0,Y 232.736,Z 478,A -85,B 0,C 180,E1 -19529.997,E2 -19529.997} C_VEL
LIN {X 0,Y 232.684,Z 478.537,A -85,B 0,C 180,E1 -19531.728,E2 -19531.728} C_VEL
LIN {X 0,Y 232.694,Z 478.503,A -85,B 0,C 180,E1 -19534.57,E2 -19534.57} C_VEL
LIN {X 0,Y 233.006,Z 477.63,A -85,B 0,C 180,E1 -19536.926,E2 -19536.926} C_VEL
LIN {X 0,Y 233.364,Z 476.546,A -85,B 0,C 180,E1 -19538.657,E2 -19538.657} C_VEL
LIN {X 0,Y 233.863,Z 475.02,A -85,B 0,C 180,E1 -19540.385,E2 -19540.385} C_VEL
LIN {X 0,Y 234.946,Z 471.952,A -85,B 0,C 180,E1 -19542.961,E2 -19542.961} C_VEL
LIN {X 0,Y 236.414,Z 467.846,A -85,B 0,C 180,E1 -19545.515,E2 -19545.515} C_VEL
LIN {X 0,Y 238.966,Z 461.562,A -85,B 0,C 180,E1 -19548.427,E2 -19548.427} C_VEL
LIN {X 0,Y 241.607,Z 454.411,A -85,B 0,C 180,E1 -19550.998,E2 -19550.998} C_VEL
LIN {X 0,Y 244.277,Z 446.377,A -85,B 0,C 180,E1 -19553.3,E2 -19553.3} C_VEL
LIN {X 0,Y 247.042,Z 437.819,A -85,B 0,C 180,E1 -19555.257,E2 -19555.257} C_VEL
LIN {X 0,Y 249.832,Z 428.506,A -85,B 0,C 180,E1 -19556.972,E2 -19556.972} C_VEL
LIN {X 0,Y 252.849,Z 417.065,A -85,B 0,C 180,E1 -19558.647,E2 -19558.647} C_VEL
LIN {X 0,Y 255.455,Z 405.833,A -85,B 0,C 180,E1 -19559.907,E2 -19559.907} C_VEL
LIN {X 0,Y 257.678,Z 393.301,A -85,B 0,C 180,E1 -19560.981,E2 -19560.981} C_VEL
LIN {X 0,Y 259.537,Z 380.303,A -85,B 0,C 180,E1 -19561.755,E2 -19561.755} C_VEL
LIN {X 0,Y 260.738,Z 366.666,A -85,B 0,C 180,E1 -19562.275,E2 -19562.275} C_VEL
LIN {X 0,Y 263.637,Z 318.149,A -85,B 0,C 180,E1 -19563.824,E2 -19563.824} C_VEL
LIN {X 0,Y 262.552,Z 311.011,A -85,B 0,C 180,E1 -19564.37,E2 -19564.37} C_VEL
LIN {X 0,Y 257.998,Z 300.397,A -85,B 0,C 180,E1 -19565.858,E2 -19565.858} C_VEL
LIN {X 0,Y 253.145,Z 290.483,A -85,B 0,C 180,E1 -19567.521,E2 -19567.521} C_VEL
LIN {X 0,Y 247.694,Z 281.056,A -85,B 0,C 180,E1 -19569.474,E2 -19569.474} C_VEL
LIN {X 0,Y 244.379,Z 275.817,A -85,B 0,C 180,E1 -19570.766,E2 -19570.766} C_VEL
LIN {X 0,Y 240.811,Z 270.458,A -85,B 0,C 180,E1 -19572.227,E2 -19572.227} C_VEL
LIN {X 0,Y 237.33,Z 265.24,A -85,B 0,C 180,E1 -19573.885,E2 -19573.885} C_VEL
LIN {X 0,Y 236.027,Z 261.292,A -85,B 0,C 180,E1 -19576.764,E2 -19576.764} C_VEL
LIN {X 0,Y 234.909,Z 257.938,A -85,B 0,C 180,E1 -19579.675,E2 -19579.675} C_VEL
LIN {X 0,Y 234.924,Z 257.715,A -85,B 0,C 180,E1 -19583.239,E2 -19583.239} C_VEL
LIN {X 0,Y 234.959,Z 257.71,A -85,B 0,C 180,E1 -19587.414,E2 -19587.414} C_VEL
LIN {X 0,Y 234.901,Z 257.721,A -85,B 0,C 180,E1 -19591.389,E2 -19591.389} C_VEL
LIN {X 0,Y 234.955,Z 257.717,A -85,B 0,C 180,E1 -19595.233,E2 -19595.233} C_VEL
LIN {X 0,Y 234.938,Z 257.721,A -85,B 0,C 180,E1 -19598.952,E2 -19598.952} C_VEL
LIN {X 0,Y 235.047,Z 257.704,A -85,B 0,C 180,E1 -19603.087,E2 -19603.087} C_VEL
LIN {X 0,Y 235.079,Z 257.693,A -85,B 0,C 180,E1 -19607.909,E2 -19607.909} C_VEL
LIN {X 0,Y 235.296,Z 257.667,A -85,B 0,C 180,E1 -19611.4,E2 -19611.4} C_VEL
LIN {X 0,Y 235.339,Z 257.669,A -85,B 0,C 180,E1 -19613.129,E2 -19613.129} C_VEL
LIN {X 0,Y 235.585,Z 257.78,A -85,B 0,C 180,E1 -19618.707,E2 -19618.707} C_VEL
LIN {X 0,Y 236.745,Z 261.478,A -85,B 0,C 180,E1 -19621.796,E2 -19621.796} C_VEL
LIN {X 0,Y 237.483,Z 263.116,A -85,B 0,C 180,E1 -19622.374,E2 -19622.374} C_VEL
LIN {X 0,Y 241.486,Z 268.783,A -85,B 0,C 180,E1 -19624.161,E2 -19624.161} C_VEL
LIN {X 0,Y 245.048,Z 273.719,A -85,B 0,C 180,E1 -19625.583,E2 -19625.583} C_VEL
LIN {X 0,Y 248.248,Z 278.736,A -85,B 0,C 180,E1 -19626.823,E2 -19626.823} C_VEL
LIN {X 0,Y 253.295,Z 287.397,A -85,B 0,C 180,E1 -19628.625,E2 -19628.625} C_VEL
LIN {X 0,Y 258.544,Z 297.398,A -85,B 0,C 180,E1 -19630.388,E2 -19630.388} C_VEL
LIN {X 0,Y 263.506,Z 308.658,A -85,B 0,C 180,E1 -19631.987,E2 -19631.987} C_VEL
LIN {X 0,Y 264.114,Z 310.21,A -85,B 0,C 180,E1 -19632.184,E2 -19632.184} C_VEL
LIN {X 0,Y 260.234,Z 370.167,A -85,B 0,C 180,E1 -19634.105,E2 -19634.105} C_VEL
LIN {X 0,Y 258.543,Z 384.299,A -85,B 0,C 180,E1 -19634.853,E2 -19634.853} C_VEL
LIN {X 0,Y 256.662,Z 396.105,A -85,B 0,C 180,E1 -19635.778,E2 -19635.778} C_VEL
LIN {X 0,Y 254.119,Z 408.491,A -85,B 0,C 180,E1 -19637.085,E2 -19637.085} C_VEL
LIN {X 0,Y 251.407,Z 419.441,A -85,B 0,C 180,E1 -19638.577,E2 -19638.577} C_VEL
LIN {X 0,Y 248.673,Z 429.048,A -85,B 0,C 180,E1 -19640.225,E2 -19640.225} C_VEL
LIN {X 0,Y 245.922,Z 437.773,A -85,B 0,C 180,E1 -19642.089,E2 -19642.089} C_VEL
LIN {X 0,Y 243.048,Z 445.953,A -85,B 0,C 180,E1 -19644.255,E2 -19644.255} C_VEL
LIN {X 0,Y 240.097,Z 454.034,A -85,B 0,C 180,E1 -19646.967,E2 -19646.967} C_VEL
LIN {X 0,Y 237.698,Z 460.208,A -85,B 0,C 180,E1 -19649.67,E2 -19649.67} C_VEL
LIN {X 0,Y 235.798,Z 464.969,A -85,B 0,C 180,E1 -19652.429,E2 -19652.429} C_VEL
LIN {X 0,Y 234.624,Z 467.91,A -85,B 0,C 180,E1 -19654.673,E2 -19654.673} C_VEL
LIN {X 0,Y 233.667,Z 470.078,A -85,B 0,C 180,E1 -19656.963,E2 -19656.963} C_VEL
LIN {X 0,Y 232.986,Z 471.528,A -85,B 0,C 180,E1 -19659.288,E2 -19659.288} C_VEL
LIN {X 0,Y 232.576,Z 472.277,A -85,B 0,C 180,E1 -19661.648,E2 -19661.648} C_VEL
LIN {X 0,Y 232.323,Z 472.246,A -85,B 0,C 180,E1 -19664.069,E2 -19664.069} C_VEL
LIN {X 0,Y 232.256,Z 471.382,A -85,B 0,C 180,E1 -19666.551,E2 -19666.551} C_VEL
LIN {X 0,Y 232.306,Z 469.604,A -85,B 0,C 180,E1 -19669.12,E2 -19669.12} C_VEL
LIN {X 0,Y 232.69,Z 466.831,A -85,B 0,C 180,E1 -19671.723,E2 -19671.723} C_VEL
LIN {X 0,Y 233.226,Z 462.827,A -85,B 0,C 180,E1 -19674.425,E2 -19674.425} C_VEL
LIN {X 0,Y 234.049,Z 457.201,A -85,B 0,C 180,E1 -19677.286,E2 -19677.286} C_VEL
LIN {X 0,Y 235.205,Z 450.184,A -85,B 0,C 180,E1 -19680.028,E2 -19680.028} C_VEL
LIN {X 0,Y 236.678,Z 441.722,A -85,B 0,C 180,E1 -19682.633,E2 -19682.633} C_VEL
LIN {X 0,Y 238.278,Z 432.433,A -85,B 0,C 180,E1 -19684.917,E2 -19684.917} C_VEL
LIN {X 0,Y 240.051,Z 421.994,A -85,B 0,C 180,E1 -19686.951,E2 -19686.951} C_VEL
LIN {X 0,Y 241.717,Z 411.127,A -85,B 0,C 180,E1 -19688.643,E2 -19688.643} C_VEL
LIN {X 0,Y 243.369,Z 398.89,A -85,B 0,C 180,E1 -19690.124,E2 -19690.124} C_VEL
LIN {X 0,Y 244.76,Z 385.681,A -85,B 0,C 180,E1 -19691.317,E2 -19691.317} C_VEL
LIN {X 0,Y 245.865,Z 372.561,A -85,B 0,C 180,E1 -19692.134,E2 -19692.134} C_VEL
LIN {X 0,Y 246.777,Z 354.043,A -85,B 0,C 180,E1 -19692.817,E2 -19692.817} C_VEL
LIN {X 0,Y 248.803,Z 301.277,A -85,B 0,C 180,E1 -19694.521,E2 -19694.521} C_VEL
LIN {X 0,Y 247.214,Z 292.87,A -85,B 0,C 180,E1 -19694.972,E2 -19694.972} C_VEL
LIN {X 0,Y 238.813,Z 269.356,A -85,B 0,C 180,E1 -19696.676,E2 -19696.676} C_VEL
LIN {X 0,Y 235.938,Z 261.727,A -85,B 0,C 180,E1 -19697.313,E2 -19697.313} C_VEL
LIN {X 0,Y 235.566,Z 259.917,A -85,B 0,C 180,E1 -19697.949,E2 -19697.949} C_VEL
LIN {X 0,Y 235.145,Z 257.723,A -85,B 0,C 180,E1 -19699.074,E2 -19699.074} C_VEL
LIN {X 0,Y 235.314,Z 257.671,A -85,B 0,C 180,E1 -19703.142,E2 -19703.142} C_VEL
LIN {X 0,Y 235.541,Z 257.645,A -85,B 0,C 180,E1 -19708.293,E2 -19708.293} C_VEL
LIN {X 0,Y 235.542,Z 257.644,A -85,B 0,C 180,E1 -19711.713,E2 -19711.713} C_VEL
LIN {X 0,Y 235.337,Z 257.67,A -85,B 0,C 180,E1 -19716.863,E2 -19716.863} C_VEL
LIN {X 0,Y 235.176,Z 257.677,A -85,B 0,C 180,E1 -19720.332,E2 -19720.332} C_VEL
LIN {X 0,Y 235.037,Z 257.704,A -85,B 0,C 180,E1 -19725.614,E2 -19725.614} C_VEL
LIN {X 0,Y 234.948,Z 257.704,A -85,B 0,C 180,E1 -19729.214,E2 -19729.214} C_VEL
LIN {X 0,Y 234.899,Z 257.723,A -85,B 0,C 180,E1 -19732.892,E2 -19732.892} C_VEL
LIN {X 0,Y 234.917,Z 257.71,A -85,B 0,C 180,E1 -19736.667,E2 -19736.667} C_VEL
LIN {X 0,Y 234.875,Z 257.713,A -85,B 0,C 180,E1 -19740.579,E2 -19740.579} C_VEL
LIN {X 0,Y 234.917,Z 257.722,A -85,B 0,C 180,E1 -19744.643,E2 -19744.643} C_VEL
LIN {X 0,Y 234.928,Z 257.714,A -85,B 0,C 180,E1 -19748.963,E2 -19748.963} C_VEL
LIN {X 0,Y 234.951,Z 257.716,A -85,B 0,C 180,E1 -19753.475,E2 -19753.475} C_VEL
LIN {X 0,Y 234.963,Z 257.71,A -85,B 0,C 180,E1 -19756.551,E2 -19756.551} C_VEL
LIN {X 0,Y 234.958,Z 257.717,A -85,B 0,C 180,E1 -19761.104,E2 -19761.104} C_VEL
LIN {X 0,Y 234.937,Z 257.711,A -85,B 0,C 180,E1 -19765.38,E2 -19765.38} C_VEL
LIN {X 0,Y 234.903,Z 257.724,A -85,B 0,C 180,E1 -19769.444,E2 -19769.444} C_VEL
LIN {X 0,Y 234.978,Z 257.704,A -85,B 0,C 180,E1 -19773.807,E2 -19773.807} C_VEL
LIN {X 0,Y 234.945,Z 257.718,A -85,B 0,C 180,E1 -19778.977,E2 -19778.977} C_VEL
LIN {X 0,Y 235.049,Z 257.699,A -85,B 0,C 180,E1 -19783.106,E2 -19783.106} C_VEL
LIN {X 0,Y 235.108,Z 257.699,A -85,B 0,C 180,E1 -19787.934,E2 -19787.934} C_VEL
LIN {X 0,Y 235.313,Z 257.67,A -85,B 0,C 180,E1 -19791.424,E2 -19791.424} C_VEL
LIN {X 0,Y 235.351,Z 257.657,A -85,B 0,C 180,E1 -19793.152,E2 -19793.152} C_VEL
LIN {X 0,Y 235.586,Z 257.638,A -85,B 0,C 180,E1 -19798.302,E2 -19798.302} C_VEL
LIN {X 0,Y 235.587,Z 257.629,A -85,B 0,C 180,E1 -19801.721,E2 -19801.721} C_VEL
LIN {X 0,Y 235.36,Z 257.644,A -85,B 0,C 180,E1 -19806.871,E2 -19806.871} C_VEL
LIN {X 0,Y 235.226,Z 257.68,A -85,B 0,C 180,E1 -19810.338,E2 -19810.338} C_VEL
LIN {X 0,Y 235.09,Z 257.693,A -85,B 0,C 180,E1 -19815.619,E2 -19815.619} C_VEL
LIN {X 0,Y 234.984,Z 257.694,A -85,B 0,C 180,E1 -19819.218,E2 -19819.218} C_VEL
LIN {X 0,Y 234.96,Z 257.717,A -85,B 0,C 180,E1 -19822.893,E2 -19822.893} C_VEL
LIN {X 0,Y 234.977,Z 257.71,A -85,B 0,C 180,E1 -19826.458,E2 -19826.458} C_VEL
LIN {X 0,Y 234.274,Z 257.799,A -85,B 0,C 180,E1 -19827.888,E2 -19827.888} C_VEL
LIN {X 0,Y 231.443,Z 258.16,A -85,B 0,C 180,E1 -19830.223,E2 -19830.223} C_VEL
LIN {X 0,Y 228.225,Z 258.558,A -85,B 0,C 180,E1 -19833.104,E2 -19833.104} C_VEL
LIN {X 0,Y 227.879,Z 258.592,A -85,B 0,C 180,E1 -19834.102,E2 -19834.102} C_VEL
LIN {X 0,Y 227.869,Z 258.598,A -85,B 0,C 180,E1 -19838.098,E2 -19838.098} C_VEL
LIN {X 0,Y 227.8,Z 258.601,A -85,B 0,C 180,E1 -19842.757,E2 -19842.757} C_VEL
LIN {X 0,Y 227.831,Z 258.607,A -85,B 0,C 180,E1 -19845.206,E2 -19845.206} C_VEL
LIN {X 0,Y 227.854,Z 258.603,A -85,B 0,C 180,E1 -19850.467,E2 -19850.467} C_VEL
LIN {X 0,Y 227.918,Z 258.678,A -85,B 0,C 180,E1 -19854.132,E2 -19854.132} C_VEL
LIN {X 0,Y 229.718,Z 267.147,A -85,B 0,C 180,E1 -19857.955,E2 -19857.955} C_VEL
LIN {X 0,Y 231.16,Z 271.244,A -85,B 0,C 180,E1 -19858.368,E2 -19858.368} C_VEL
LIN {X 0,Y 238.983,Z 292.86,A -85,B 0,C 180,E1 -19860.035,E2 -19860.035} C_VEL
LIN {X 0,Y 241.856,Z 315.314,A -85,B 0,C 180,E1 -19861.151,E2 -19861.151} C_VEL
LIN {X 0,Y 239.378,Z 375.122,A -85,B 0,C 180,E1 -19863.164,E2 -19863.164} C_VEL
LIN {X 0,Y 238.288,Z 389.224,A -85,B 0,C 180,E1 -19863.975,E2 -19863.975} C_VEL
LIN {X 0,Y 237.013,Z 401.423,A -85,B 0,C 180,E1 -19865.002,E2 -19865.002} C_VEL
LIN {X 0,Y 235.141,Z 414.022,A -85,B 0,C 180,E1 -19866.434,E2 -19866.434} C_VEL
LIN {X 0,Y 233.344,Z 425.353,A -85,B 0,C 180,E1 -19868.114,E2 -19868.114} C_VEL
LIN {X 0,Y 231.666,Z 435.606,A -85,B 0,C 180,E1 -19870.043,E2 -19870.043} C_VEL
LIN {X 0,Y 230.087,Z 444.851,A -85,B 0,C 180,E1 -19872.212,E2 -19872.212} C_VEL
LIN {X 0,Y 228.44,Z 453.853,A -85,B 0,C 180,E1 -19874.838,E2 -19874.838} C_VEL
LIN {X 0,Y 227.153,Z 461.018,A -85,B 0,C 180,E1 -19877.489,E2 -19877.489} C_VEL
LIN {X 0,Y 226.36,Z 466.728,A -85,B 0,C 180,E1 -19880.165,E2 -19880.165} C_VEL
LIN {X 0,Y 225.852,Z 471.182,A -85,B 0,C 180,E1 -19882.847,E2 -19882.847} C_VEL
LIN {X 0,Y 225.612,Z 474.512,A -85,B 0,C 180,E1 -19885.531,E2 -19885.531} C_VEL
LIN {X 0,Y 225.588,Z 476.813,A -85,B 0,C 180,E1 -19888.212,E2 -19888.212} C_VEL
LIN {X 0,Y 225.652,Z 477.799,A -85,B 0,C 180,E1 -19889.997,E2 -19889.997} C_VEL
LIN {X 0,Y 225.584,Z 478.379,A -85,B 0,C 180,E1 -19891.782,E2 -19891.782} C_VEL
LIN {X 0,Y 225.61,Z 478.458,A -85,B 0,C 180,E1 -19894.463,E2 -19894.463} C_VEL
LIN {X 0,Y 225.951,Z 477.64,A -85,B 0,C 180,E1 -19897.144,E2 -19897.144} C_VEL
LIN {X 0,Y 226.33,Z 476.603,A -85,B 0,C 180,E1 -19898.929,E2 -19898.929} C_VEL
LIN {X 0,Y 226.867,Z 475.164,A -85,B 0,C 180,E1 -19900.709,E2 -19900.709} C_VEL
LIN {X 0,Y 228.025,Z 472.176,A -85,B 0,C 180,E1 -19903.362,E2 -19903.362} C_VEL
LIN {X 0,Y 229.577,Z 468.162,A -85,B 0,C 180,E1 -19905.989,E2 -19905.989} C_VEL
LIN {X 0,Y 232.252,Z 462.018,A -85,B 0,C 180,E1 -19908.98,E2 -19908.98} C_VEL
LIN {X 0,Y 234.99,Z 455.128,A -85,B 0,C 180,E1 -19911.581,E2 -19911.581} C_VEL
LIN {X 0,Y 237.276,Z 448.668,A -85,B 0,C 180,E1 -19913.566,E2 -19913.566} C_VEL
LIN {X 0,Y 240.058,Z 440.624,A -85,B 0,C 180,E1 -19915.58,E2 -19915.58} C_VEL
LIN {X 0,Y 243.27,Z 430.854,A -85,B 0,C 180,E1 -19917.528,E2 -19917.528} C_VEL
LIN {X 0,Y 246.37,Z 420.004,A -85,B 0,C 180,E1 -19919.239,E2 -19919.239} C_VEL
LIN {X 0,Y 248.997,Z 409.514,A -85,B 0,C 180,E1 -19920.531,E2 -19920.531} C_VEL
LIN {X 0,Y 251.736,Z 396.142,A -85,B 0,C 180,E1 -19921.796,E2 -19921.796} C_VEL
LIN {X 0,Y 253.762,Z 383.567,A -85,B 0,C 180,E1 -19922.625,E2 -19922.625} C_VEL
LIN {X 0,Y 255.261,Z 369.558,A -85,B 0,C 180,E1 -19923.231,E2 -19923.231} C_VEL
LIN {X 0,Y 258.469,Z 319.461,A -85,B 0,C 180,E1 -19924.856,E2 -19924.856} C_VEL
LIN {X 0,Y 257.588,Z 313.948,A -85,B 0,C 180,E1 -19925.308,E2 -19925.308} C_VEL
LIN {X 0,Y 252.678,Z 302.503,A -85,B 0,C 180,E1 -19927.023,E2 -19927.023} C_VEL
LIN {X 0,Y 248.178,Z 293.527,A -85,B 0,C 180,E1 -19928.664,E2 -19928.664} C_VEL
LIN {X 0,Y 243.577,Z 285.43,A -85,B 0,C 180,E1 -19930.451,E2 -19930.451} C_VEL
LIN {X 0,Y 240.866,Z 281.077,A -85,B 0,C 180,E1 -19931.56,E2 -19931.56} C_VEL
LIN {X 0,Y 237.626,Z 276.033,A -85,B 0,C 180,E1 -19932.981,E2 -19932.981} C_VEL
LIN {X 0,Y 233.585,Z 270.233,A -85,B 0,C 180,E1 -19934.89,E2 -19934.89} C_VEL
LIN {X 0,Y 230.308,Z 265.663,A -85,B 0,C 180,E1 -19936.627,E2 -19936.627} C_VEL
LIN {X 0,Y 229.803,Z 264.541,A -85,B 0,C 180,E1 -19937.216,E2 -19937.216} C_VEL
LIN {X 0,Y 228.744,Z 261.225,A -85,B 0,C 180,E1 -19940.179,E2 -19940.179} C_VEL
LIN {X 0,Y 227.878,Z 258.622,A -85,B 0,C 180,E1 -19943.182,E2 -19943.182} C_VEL
LIN {X 0,Y 227.886,Z 258.591,A -85,B 0,C 180,E1 -19946.368,E2 -19946.368} C_VEL
LIN {X 0,Y 227.878,Z 258.59,A -85,B 0,C 180,E1 -19950.421,E2 -19950.421} C_VEL
LIN {X 0,Y 227.905,Z 258.588,A -85,B 0,C 180,E1 -19954.412,E2 -19954.412} C_VEL
LIN {X 0,Y 227.924,Z 258.587,A -85,B 0,C 180,E1 -19958.272,E2 -19958.272} C_VEL
LIN {X 0,Y 227.997,Z 258.576,A -85,B 0,C 180,E1 -19963.882,E2 -19963.882} C_VEL
LIN {X 0,Y 228.118,Z 258.569,A -85,B 0,C 180,E1 -19969.336,E2 -19969.336} C_VEL
LIN {X 0,Y 228.291,Z 258.549,A -85,B 0,C 180,E1 -19972.915,E2 -19972.915} C_VEL
LIN {X 0,Y 228.185,Z 258.789,A -85,B 0,C 180,E1 -19975.573,E2 -19975.573} C_VEL
LIN {X 0,Y 229.744,Z 262.043,A -85,B 0,C 180,E1 -19979.003,E2 -19979.003} C_VEL
LIN {X 0,Y 233.128,Z 266.835,A -85,B 0,C 180,E1 -19980.944,E2 -19980.944} C_VEL
LIN {X 0,Y 234.738,Z 269.231,A -85,B 0,C 180,E1 -19981.758,E2 -19981.758} C_VEL
LIN {X 0,Y 238.635,Z 274.857,A -85,B 0,C 180,E1 -19983.569,E2 -19983.569} C_VEL
LIN {X 0,Y 241.924,Z 279.579,A -85,B 0,C 180,E1 -19984.956,E2 -19984.956} C_VEL
LIN {X 0,Y 245.165,Z 284.79,A -85,B 0,C 180,E1 -19986.259,E2 -19986.259} C_VEL
LIN {X 0,Y 250.75,Z 294.77,A -85,B 0,C 180,E1 -19988.351,E2 -19988.351} C_VEL
LIN {X 0,Y 256.071,Z 305.85,A -85,B 0,C 180,E1 -19990.231,E2 -19990.231} C_VEL
LIN {X 0,Y 258.864,Z 312.536,A -85,B 0,C 180,E1 -19991.172,E2 -19991.172} C_VEL
LIN {X 0,Y 254.937,Z 370.236,A -85,B 0,C 180,E1 -19993.054,E2 -19993.054} C_VEL
LIN {X 0,Y 253.194,Z 384.23,A -85,B 0,C 180,E1 -19993.807,E2 -19993.807} C_VEL
LIN {X 0,Y 251.096,Z 396.533,A -85,B 0,C 180,E1 -19994.785,E2 -19994.785} C_VEL
LIN {X 0,Y 248.345,Z 409.228,A -85,B 0,C 180,E1 -19996.166,E2 -19996.166} C_VEL
LIN {X 0,Y 245.505,Z 420.038,A -85,B 0,C 180,E1 -19997.673,E2 -19997.673} C_VEL
LIN {X 0,Y 242.493,Z 430.057,A -85,B 0,C 180,E1 -19999.456,E2 -19999.456} C_VEL
LIN {X 0,Y 239.278,Z 439.515,A -85,B 0,C 180,E1 -20001.574,E2 -20001.574} C_VEL
LIN {X 0,Y 236.21,Z 447.727,A -85,B 0,C 180,E1 -20003.887,E2 -20003.887} C_VEL
LIN {X 0,Y 233.61,Z 454.388,A -85,B 0,C 180,E1 -20006.257,E2 -20006.257} C_VEL
LIN {X 0,Y 230.977,Z 460.639,A -85,B 0,C 180,E1 -20009.118,E2 -20009.118} C_VEL
LIN {X 0,Y 229.329,Z 464.519,A -85,B 0,C 180,E1 -20011.382,E2 -20011.382} C_VEL
LIN {X 0,Y 227.404,Z 468.799,A -85,B 0,C 180,E1 -20014.855,E2 -20014.855} C_VEL
LIN {X 0,Y 226.103,Z 471.455,A -85,B 0,C 180,E1 -20018.42,E2 -20018.42} C_VEL
LIN {X 0,Y 225.482,Z 472.405,A -85,B 0,C 180,E1 -20021.584,E2 -20021.584} C_VEL
LIN {X 0,Y 225.216,Z 472.283,A -85,B 0,C 180,E1 -20024.138,E2 -20024.138} C_VEL
LIN {X 0,Y 225.152,Z 471.347,A -85,B 0,C 180,E1 -20026.634,E2 -20026.634} C_VEL
LIN {X 0,Y 225.216,Z 469.649,A -85,B 0,C 180,E1 -20029.061,E2 -20029.061} C_VEL
LIN {X 0,Y 225.548,Z 467.205,A -85,B 0,C 180,E1 -20031.455,E2 -20031.455} C_VEL
LIN {X 0,Y 226.034,Z 463.827,A -85,B 0,C 180,E1 -20033.915,E2 -20033.915} C_VEL
LIN {X 0,Y 226.788,Z 458.651,A -85,B 0,C 180,E1 -20036.767,E2 -20036.767} C_VEL
LIN {X 0,Y 227.895,Z 451.805,A -85,B 0,C 180,E1 -20039.68,E2 -20039.68} C_VEL
LIN {X 0,Y 229.208,Z 444.554,A -85,B 0,C 180,E1 -20042.126,E2 -20042.126} C_VEL
LIN {X 0,Y 230.78,Z 435.676,A -85,B 0,C 180,E1 -20044.526,E2 -20044.526} C_VEL
LIN {X 0,Y 232.521,Z 425.897,A -85,B 0,C 180,E1 -20046.649,E2 -20046.649} C_VEL
LIN {X 0,Y 234.225,Z 415.765,A -85,B 0,C 180,E1 -20048.42,E2 -20048.42} C_VEL
LIN {X 0,Y 235.837,Z 404.693,A -85,B 0,C 180,E1 -20049.962,E2 -20049.962} C_VEL
LIN {X 0,Y 237.383,Z 392.267,A -85,B 0,C 180,E1 -20051.287,E2 -20051.287} C_VEL
LIN {X 0,Y 238.683,Z 378.91,A -85,B 0,C 180,E1 -20052.326,E2 -20052.326} C_VEL
LIN {X 0,Y 239.596,Z 365.251,A -85,B 0,C 180,E1 -20053.006,E2 -20053.006} C_VEL
LIN {X 0,Y 242.168,Z 302.146,A -85,B 0,C 180,E1 -20055.108,E2 -20055.108} C_VEL
LIN {X 0,Y 240.813,Z 294.96,A -85,B 0,C 180,E1 -20055.508,E2 -20055.508} C_VEL
LIN {X 0,Y 232.093,Z 270.519,A -85,B 0,C 180,E1 -20057.349,E2 -20057.349} C_VEL
LIN {X 0,Y 228.715,Z 261.632,A -85,B 0,C 180,E1 -20058.14,E2 -20058.14} C_VEL
LIN {X 0,Y 228.156,Z 258.842,A -85,B 0,C 180,E1 -20059.353,E2 -20059.353} C_VEL
LIN {X 0,Y 228.184,Z 258.561,A -85,B 0,C 180,E1 -20060.17,E2 -20060.17} C_VEL
LIN {X 0,Y 228.266,Z 258.548,A -85,B 0,C 180,E1 -20062.929,E2 -20062.929} C_VEL
LIN {X 0,Y 228.501,Z 258.522,A -85,B 0,C 180,E1 -20068.241,E2 -20068.241} C_VEL
LIN {X 0,Y 228.501,Z 258.521,A -85,B 0,C 180,E1 -20071.766,E2 -20071.766} C_VEL
LIN {X 0,Y 228.287,Z 258.549,A -85,B 0,C 180,E1 -20077.076,E2 -20077.076} C_VEL
LIN {X 0,Y 228.097,Z 258.558,A -85,B 0,C 180,E1 -20080.656,E2 -20080.656} C_VEL
LIN {X 0,Y 227.987,Z 258.579,A -85,B 0,C 180,E1 -20086.11,E2 -20086.11} C_VEL
LIN {X 0,Y 227.88,Z 258.588,A -85,B 0,C 180,E1 -20089.834,E2 -20089.834} C_VEL
LIN {X 0,Y 227.854,Z 258.604,A -85,B 0,C 180,E1 -20093.642,E2 -20093.642} C_VEL
LIN {X 0,Y 227.829,Z 258.585,A -85,B 0,C 180,E1 -20097.565,E2 -20097.565} C_VEL
LIN {X 0,Y 227.823,Z 258.595,A -85,B 0,C 180,E1 -20101.633,E2 -20101.633} C_VEL
LIN {X 0,Y 227.858,Z 258.602,A -85,B 0,C 180,E1 -20105.879,E2 -20105.879} C_VEL
LIN {X 0,Y 227.857,Z 258.598,A -85,B 0,C 180,E1 -20110.373,E2 -20110.373} C_VEL
LIN {X 0,Y 227.883,Z 258.594,A -85,B 0,C 180,E1 -20114.84,E2 -20114.84} C_VEL
LIN {X 0,Y 227.906,Z 258.588,A -85,B 0,C 180,E1 -20117.743,E2 -20117.743} C_VEL
LIN {X 0,Y 227.864,Z 258.599,A -85,B 0,C 180,E1 -20121.931,E2 -20121.931} C_VEL
LIN {X 0,Y 227.867,Z 258.591,A -85,B 0,C 180,E1 -20126.386,E2 -20126.386} C_VEL
LIN {X 0,Y 227.885,Z 258.597,A -85,B 0,C 180,E1 -20130.449,E2 -20130.449} C_VEL
LIN {X 0,Y 227.91,Z 258.584,A -85,B 0,C 180,E1 -20134.438,E2 -20134.438} C_VEL
LIN {X 0,Y 227.922,Z 258.591,A -85,B 0,C 180,E1 -20138.297,E2 -20138.297} C_VEL
LIN {X 0,Y 228.012,Z 258.572,A -85,B 0,C 180,E1 -20143.908,E2 -20143.908} C_VEL
LIN {X 0,Y 228.063,Z 258.576,A -85,B 0,C 180,E1 -20147.555,E2 -20147.555} C_VEL
LIN {X 0,Y 228.254,Z 258.548,A -85,B 0,C 180,E1 -20151.156,E2 -20151.156} C_VEL
LIN {X 0,Y 228.304,Z 258.534,A -85,B 0,C 180,E1 -20152.939,E2 -20152.939} C_VEL
LIN {X 0,Y 228.544,Z 258.516,A -85,B 0,C 180,E1 -20158.25,E2 -20158.25} C_VEL
LIN {X 0,Y 228.545,Z 258.504,A -85,B 0,C 180,E1 -20161.774,E2 -20161.774} C_VEL
LIN {X 0,Y 228.312,Z 258.523,A -85,B 0,C 180,E1 -20167.084,E2 -20167.084} C_VEL
LIN {X 0,Y 228.157,Z 258.563,A -85,B 0,C 180,E1 -20170.662,E2 -20170.662} C_VEL
LIN {X 0,Y 228.05,Z 258.578,A -85,B 0,C 180,E1 -20174.284,E2 -20174.284} C_VEL
LIN {X 0,Y 227.947,Z 258.57,A -85,B 0,C 180,E1 -20177.969,E2 -20177.969} C_VEL
LIN {X 0,Y 227.926,Z 258.589,A -85,B 0,C 180,E1 -20182.32,E2 -20182.32} C_VEL
LIN {X 0,Y 227.946,Z 258.586,A -85,B 0,C 180,E1 -20186.599,E2 -20186.599} C_VEL
LIN {X 0,Y 227.896,Z 258.588,A -85,B 0,C 180,E1 -20190.286,E2 -20190.286} C_VEL
LIN {X 0,Y 227.879,Z 258.592,A -85,B 0,C 180,E1 -20194.102,E2 -20194.102} C_VEL
LIN {X 0,Y 227.167,Z 258.678,A -85,B 0,C 180,E1 -20195.576,E2 -20195.576} C_VEL
LIN {X 0,Y 224.316,Z 259.04,A -85,B 0,C 180,E1 -20197.982,E2 -20197.982} C_VEL
LIN {X 0,Y 221.908,Z 259.342,A -85,B 0,C 180,E1 -20199.945,E2 -20199.945} C_VEL
LIN {X 0,Y 220.859,Z 259.467,A -85,B 0,C 180,E1 -20201.468,E2 -20201.468} C_VEL
LIN {X 0,Y 220.763,Z 259.476,A -85,B 0,C 180,E1 -20201.985,E2 -20201.985} C_VEL
LIN {X 0,Y 220.774,Z 259.482,A -85,B 0,C 180,E1 -20205.542,E2 -20205.542} C_VEL
LIN {X 0,Y 220.808,Z 259.48,A -85,B 0,C 180,E1 -20210.46,E2 -20210.46} C_VEL
LIN {X 0,Y 220.896,Z 259.614,A -85,B 0,C 180,E1 -20213.657,E2 -20213.657} C_VEL
LIN {X 0,Y 222.486,Z 267.168,A -85,B 0,C 180,E1 -20217.142,E2 -20217.142} C_VEL
LIN {X 0,Y 225.169,Z 274.35,A -85,B 0,C 180,E1 -20217.827,E2 -20217.827} C_VEL
LIN {X 0,Y 232.572,Z 294.91,A -85,B 0,C 180,E1 -20219.451,E2 -20219.451} C_VEL
LIN {X 0,Y 235.251,Z 315.387,A -85,B 0,C 180,E1 -20220.516,E2 -20220.516} C_VEL
LIN {X 0,Y 232.719,Z 374.886,A -85,B 0,C 180,E1 -20222.575,E2 -20222.575} C_VEL
LIN {X 0,Y 231.598,Z 389.02,A -85,B 0,C 180,E1 -20223.407,E2 -20223.407} C_VEL
LIN {X 0,Y 230.283,Z 401.244,A -85,B 0,C 180,E1 -20224.461,E2 -20224.461} C_VEL
LIN {X 0,Y 228.348,Z 413.861,A -85,B 0,C 180,E1 -20225.93,E2 -20225.93} C_VEL
LIN {X 0,Y 226.502,Z 425.206,A -85,B 0,C 180,E1 -20227.657,E2 -20227.657} C_VEL
LIN {X 0,Y 224.766,Z 435.47,A -85,B 0,C 180,E1 -20229.641,E2 -20229.641} C_VEL
LIN {X 0,Y 222.944,Z 445.555,A -85,B 0,C 180,E1 -20232.097,E2 -20232.097} C_VEL
LIN {X 0,Y 221.298,Z 454.399,A -85,B 0,C 180,E1 -20234.808,E2 -20234.808} C_VEL
LIN {X 0,Y 220.037,Z 461.421,A -85,B 0,C 180,E1 -20237.547,E2 -20237.547} C_VEL
LIN {X 0,Y 219.119,Z 467.851,A -85,B 0,C 180,E1 -20240.769,E2 -20240.769} C_VEL
LIN {X 0,Y 218.666,Z 472.016,A -85,B 0,C 180,E1 -20243.538,E2 -20243.538} C_VEL
LIN {X 0,Y 218.482,Z 475.075,A -85,B 0,C 180,E1 -20246.308,E2 -20246.308} C_VEL
LIN {X 0,Y 218.491,Z 476.556,A -85,B 0,C 180,E1 -20248.154,E2 -20248.154} C_VEL
LIN {X 0,Y 218.571,Z 477.586,A -85,B 0,C 180,E1 -20249.997,E2 -20249.997} C_VEL
LIN {X 0,Y 218.487,Z 478.209,A -85,B 0,C 180,E1 -20251.84,E2 -20251.84} C_VEL
LIN {X 0,Y 218.51,Z 478.413,A -85,B 0,C 180,E1 -20254.286,E2 -20254.286} C_VEL
LIN {X 0,Y 218.889,Z 477.652,A -85,B 0,C 180,E1 -20257.376,E2 -20257.376} C_VEL
LIN {X 0,Y 219.888,Z 475.275,A -85,B 0,C 180,E1 -20261.053,E2 -20261.053} C_VEL
LIN {X 0,Y 221.118,Z 472.379,A -85,B 0,C 180,E1 -20263.787,E2 -20263.787} C_VEL
LIN {X 0,Y 222.764,Z 468.485,A -85,B 0,C 180,E1 -20266.492,E2 -20266.492} C_VEL
LIN {X 0,Y 225.181,Z 463.47,A -85,B 0,C 180,E1 -20269.126,E2 -20269.126} C_VEL
LIN {X 0,Y 227.899,Z 457.211,A -85,B 0,C 180,E1 -20271.716,E2 -20271.716} C_VEL
LIN {X 0,Y 230.283,Z 450.865,A -85,B 0,C 180,E1 -20273.848,E2 -20273.848} C_VEL
LIN {X 0,Y 233.118,Z 443.28,A -85,B 0,C 180,E1 -20275.918,E2 -20275.918} C_VEL
LIN {X 0,Y 236.719,Z 433.119,A -85,B 0,C 180,E1 -20278.116,E2 -20278.116} C_VEL
LIN {X 0,Y 240.326,Z 421.61,A -85,B 0,C 180,E1 -20280.049,E2 -20280.049} C_VEL
LIN {X 0,Y 243.426,Z 409.983,A -85,B 0,C 180,E1 -20281.549,E2 -20281.549} C_VEL
LIN {X 0,Y 246.065,Z 397.822,A -85,B 0,C 180,E1 -20282.74,E2 -20282.74} C_VEL
LIN {X 0,Y 248.412,Z 384.545,A -85,B 0,C 180,E1 -20283.661,E2 -20283.661} C_VEL
LIN {X 0,Y 249.98,Z 370.897,A -85,B 0,C 180,E1 -20284.283,E2 -20284.283} C_VEL
LIN {X 0,Y 253.377,Z 320.805,A -85,B 0,C 180,E1 -20285.934,E2 -20285.934} C_VEL
LIN {X 0,Y 252.787,Z 317.209,A -85,B 0,C 180,E1 -20286.256,E2 -20286.256} C_VEL
LIN {X 0,Y 248.32,Z 306.513,A -85,B 0,C 180,E1 -20287.933,E2 -20287.933} C_VEL
LIN {X 0,Y 244.375,Z 298.471,A -85,B 0,C 180,E1 -20289.457,E2 -20289.457} C_VEL
LIN {X 0,Y 240.023,Z 290.586,A -85,B 0,C 180,E1 -20291.256,E2 -20291.256} C_VEL
LIN {X 0,Y 237.314,Z 286.155,A -85,B 0,C 180,E1 -20292.428,E2 -20292.428} C_VEL
LIN {X 0,Y 234.509,Z 281.634,A -85,B 0,C 180,E1 -20293.746,E2 -20293.746} C_VEL
LIN {X 0,Y 231.056,Z 276.417,A -85,B 0,C 180,E1 -20295.475,E2 -20295.475} C_VEL
LIN {X 0,Y 227.745,Z 271.722,A -85,B 0,C 180,E1 -20297.305,E2 -20297.305} C_VEL
LIN {X 0,Y 223.587,Z 266.335,A -85,B 0,C 180,E1 -20299.911,E2 -20299.911} C_VEL
LIN {X 0,Y 222.579,Z 264.575,A -85,B 0,C 180,E1 -20300.827,E2 -20300.827} C_VEL
LIN {X 0,Y 221.904,Z 262.544,A -85,B 0,C 180,E1 -20302.992,E2 -20302.992} C_VEL
LIN {X 0,Y 220.829,Z 259.529,A -85,B 0,C 180,E1 -20307.37,E2 -20307.37} C_VEL
LIN {X 0,Y 220.806,Z 259.477,A -85,B 0,C 180,E1 -20311.471,E2 -20311.471} C_VEL
LIN {X 0,Y 220.847,Z 259.477,A -85,B 0,C 180,E1 -20315.551,E2 -20315.551} C_VEL
LIN {X 0,Y 220.848,Z 259.472,A -85,B 0,C 180,E1 -20319.498,E2 -20319.498} C_VEL
LIN {X 0,Y 220.963,Z 259.455,A -85,B 0,C 180,E1 -20323.355,E2 -20323.355} C_VEL
LIN {X 0,Y 221.043,Z 259.446,A -85,B 0,C 180,E1 -20328.991,E2 -20328.991} C_VEL
LIN {X 0,Y 221.23,Z 259.667,A -85,B 0,C 180,E1 -20331.54,E2 -20331.54} C_VEL
LIN {X 0,Y 222.221,Z 262.488,A -85,B 0,C 180,E1 -20335.113,E2 -20335.113} C_VEL
LIN {X 0,Y 224.859,Z 266.099,A -85,B 0,C 180,E1 -20337.03,E2 -20337.03} C_VEL
LIN {X 0,Y 227.502,Z 268.733,A -85,B 0,C 180,E1 -20338.606,E2 -20338.606} C_VEL
LIN {X 0,Y 231.578,Z 274.469,A -85,B 0,C 180,E1 -20340.868,E2 -20340.868} C_VEL
LIN {X 0,Y 235.97,Z 281.15,A -85,B 0,C 180,E1 -20343.03,E2 -20343.03} C_VEL
LIN {X 0,Y 238.981,Z 285.639,A -85,B 0,C 180,E1 -20344.374,E2 -20344.374} C_VEL
LIN {X 0,Y 241.902,Z 290.459,A -85,B 0,C 180,E1 -20345.597,E2 -20345.597} C_VEL
LIN {X 0,Y 247.206,Z 300.361,A -85,B 0,C 180,E1 -20347.709,E2 -20347.709} C_VEL
LIN {X 0,Y 251.859,Z 310.368,A -85,B 0,C 180,E1 -20349.437,E2 -20349.437} C_VEL
LIN {X 0,Y 253.706,Z 314.954,A -85,B 0,C 180,E1 -20350.121,E2 -20350.121} C_VEL
LIN {X 0,Y 249.75,Z 370.399,A -85,B 0,C 180,E1 -20351.959,E2 -20351.959} C_VEL
LIN {X 0,Y 247.961,Z 384.04,A -85,B 0,C 180,E1 -20352.693,E2 -20352.693} C_VEL
LIN {X 0,Y 245.875,Z 396.018,A -85,B 0,C 180,E1 -20353.644,E2 -20353.644} C_VEL
LIN {X 0,Y 243.335,Z 407.5,A -85,B 0,C 180,E1 -20354.873,E2 -20354.873} C_VEL
LIN {X 0,Y 240.258,Z 418.762,A -85,B 0,C 180,E1 -20356.417,E2 -20356.417} C_VEL
LIN {X 0,Y 236.885,Z 429.54,A -85,B 0,C 180,E1 -20358.318,E2 -20358.318} C_VEL
LIN {X 0,Y 233.248,Z 439.686,A -85,B 0,C 180,E1 -20360.63,E2 -20360.63} C_VEL
LIN {X 0,Y 230.239,Z 447.319,A -85,B 0,C 180,E1 -20362.809,E2 -20362.809} C_VEL
LIN {X 0,Y 226.951,Z 455.179,A -85,B 0,C 180,E1 -20365.677,E2 -20365.677} C_VEL
LIN {X 0,Y 224.178,Z 461.309,A -85,B 0,C 180,E1 -20368.63,E2 -20368.63} C_VEL
LIN {X 0,Y 222.191,Z 465.588,A -85,B 0,C 180,E1 -20371.355,E2 -20371.355} C_VEL
LIN {X 0,Y 220.204,Z 469.64,A -85,B 0,C 180,E1 -20375.046,E2 -20375.046} C_VEL
LIN {X 0,Y 219.267,Z 471.342,A -85,B 0,C 180,E1 -20377.498,E2 -20377.498} C_VEL
LIN {X 0,Y 218.631,Z 472.301,A -85,B 0,C 180,E1 -20379.99,E2 -20379.99} C_VEL
LIN {X 0,Y 218.262,Z 472.547,A -85,B 0,C 180,E1 -20382.527,E2 -20382.527} C_VEL
LIN {X 0,Y 218.073,Z 472.015,A -85,B 0,C 180,E1 -20385.133,E2 -20385.133} C_VEL
LIN {X 0,Y 218.032,Z 470.582,A -85,B 0,C 180,E1 -20387.826,E2 -20387.826} C_VEL
LIN {X 0,Y 218.301,Z 468.2,A -85,B 0,C 180,E1 -20390.569,E2 -20390.569} C_VEL
LIN {X 0,Y 218.817,Z 464.713,A -85,B 0,C 180,E1 -20393.387,E2 -20393.387} C_VEL
LIN {X 0,Y 219.534,Z 459.86,A -85,B 0,C 180,E1 -20396.312,E2 -20396.312} C_VEL
LIN {X 0,Y 220.624,Z 453.201,A -85,B 0,C 180,E1 -20399.362,E2 -20399.362} C_VEL
LIN {X 0,Y 222.163,Z 444.927,A -85,B 0,C 180,E1 -20402.312,E2 -20402.312} C_VEL
LIN {X 0,Y 223.678,Z 436.649,A -85,B 0,C 180,E1 -20404.66,E2 -20404.66} C_VEL
LIN {X 0,Y 225.39,Z 427.193,A -85,B 0,C 180,E1 -20406.821,E2 -20406.821} C_VEL
LIN {X 0,Y 227.195,Z 417.021,A -85,B 0,C 180,E1 -20408.69,E2 -20408.69} C_VEL
LIN {X 0,Y 228.967,Z 405.35,A -85,B 0,C 180,E1 -20410.398,E2 -20410.398} C_VEL
LIN {X 0,Y 230.651,Z 392.46,A -85,B 0,C 180,E1 -20411.817,E2 -20411.817} C_VEL
LIN {X 0,Y 231.975,Z 379.235,A -85,B 0,C 180,E1 -20412.88,E2 -20412.88} C_VEL
LIN {X 0,Y 232.934,Z 365.807,A -85,B 0,C 180,E1 -20413.573,E2 -20413.573} C_VEL
LIN {X 0,Y 235.542,Z 302.77,A -85,B 0,C 180,E1 -20415.739,E2 -20415.739} C_VEL
LIN {X 0,Y 234.443,Z 297.133,A -85,B 0,C 180,E1 -20416.068,E2 -20416.068} C_VEL
LIN {X 0,Y 225.842,Z 272.987,A -85,B 0,C 180,E1 -20417.955,E2 -20417.955} C_VEL
LIN {X 0,Y 221.532,Z 261.727,A -85,B 0,C 180,E1 -20418.983,E2 -20418.983} C_VEL
LIN {X 0,Y 221.159,Z 259.577,A -85,B 0,C 180,E1 -20419.943,E2 -20419.943} C_VEL
LIN {X 0,Y 221.203,Z 259.427,A -85,B 0,C 180,E1 -20422.702,E2 -20422.702} C_VEL
LIN {X 0,Y 221.459,Z 259.399,A -85,B 0,C 180,E1 -20428.185,E2 -20428.185} C_VEL
LIN {X 0,Y 221.46,Z 259.398,A -85,B 0,C 180,E1 -20431.822,E2 -20431.822} C_VEL
LIN {X 0,Y 221.222,Z 259.43,A -85,B 0,C 180,E1 -20437.304,E2 -20437.304} C_VEL
LIN {X 0,Y 221.027,Z 259.439,A -85,B 0,C 180,E1 -20441.001,E2 -20441.001} C_VEL
LIN {X 0,Y 220.951,Z 259.454,A -85,B 0,C 180,E1 -20446.638,E2 -20446.638} C_VEL
LIN {X 0,Y 220.829,Z 259.471,A -85,B 0,C 180,E1 -20450.495,E2 -20450.495} C_VEL
LIN {X 0,Y 220.811,Z 259.476,A -85,B 0,C 180,E1 -20454.445,E2 -20454.445} C_VEL
LIN {X 0,Y 220.778,Z 259.453,A -85,B 0,C 180,E1 -20458.525,E2 -20458.525} C_VEL
LIN {X 0,Y 220.778,Z 259.48,A -85,B 0,C 180,E1 -20462.766,E2 -20462.766} C_VEL
LIN {X 0,Y 220.799,Z 259.477,A -85,B 0,C 180,E1 -20467.299,E2 -20467.299} C_VEL
LIN {X 0,Y 220.823,Z 259.477,A -85,B 0,C 180,E1 -20471.943,E2 -20471.943} C_VEL
LIN {X 0,Y 220.84,Z 259.469,A -85,B 0,C 180,E1 -20475.584,E2 -20475.584} C_VEL
LIN {X 0,Y 220.837,Z 259.473,A -85,B 0,C 180,E1 -20479.803,E2 -20479.803} C_VEL
LIN {X 0,Y 220.818,Z 259.476,A -85,B 0,C 180,E1 -20482.81,E2 -20482.81} C_VEL
LIN {X 0,Y 220.801,Z 259.478,A -85,B 0,C 180,E1 -20487.258,E2 -20487.258} C_VEL
LIN {X 0,Y 220.809,Z 259.477,A -85,B 0,C 180,E1 -20491.498,E2 -20491.498} C_VEL
LIN {X 0,Y 220.847,Z 259.467,A -85,B 0,C 180,E1 -20495.578,E2 -20495.578} C_VEL
LIN {X 0,Y 220.849,Z 259.475,A -85,B 0,C 180,E1 -20499.524,E2 -20499.524} C_VEL
LIN {X 0,Y 220.97,Z 259.45,A -85,B 0,C 180,E1 -20503.38,E2 -20503.38} C_VEL
LIN {X 0,Y 220.999,Z 259.453,A -85,B 0,C 180,E1 -20507.151,E2 -20507.151} C_VEL
LIN {X 0,Y 221.195,Z 259.427,A -85,B 0,C 180,E1 -20510.872,E2 -20510.872} C_VEL
LIN {X 0,Y 221.12,Z 259.436,A -85,B 0,C 180,E1 -20514.541,E2 -20514.541} C_VEL
LIN {X 0,Y 221.478,Z 259.396,A -85,B 0,C 180,E1 -20518.194,E2 -20518.194} C_VEL
LIN {X 0,Y 221.478,Z 259.382,A -85,B 0,C 180,E1 -20521.83,E2 -20521.83} C_VEL
LIN {X 0,Y 221.25,Z 259.404,A -85,B 0,C 180,E1 -20527.311,E2 -20527.311} C_VEL
LIN {X 0,Y 221.078,Z 259.445,A -85,B 0,C 180,E1 -20531.007,E2 -20531.007} C_VEL
LIN {X 0,Y 220.996,Z 259.441,A -85,B 0,C 180,E1 -20536.643,E2 -20536.643} C_VEL
LIN {X 0,Y 220.873,Z 259.456,A -85,B 0,C 180,E1 -20540.499,E2 -20540.499} C_VEL
LIN {X 0,Y 220.869,Z 259.473,A -85,B 0,C 180,E1 -20544.446,E2 -20544.446} C_VEL
LIN {X 0,Y 220.826,Z 259.461,A -85,B 0,C 180,E1 -20548.526,E2 -20548.526} C_VEL
LIN {X 0,Y 220.839,Z 259.476,A -85,B 0,C 180,E1 -20552.764,E2 -20552.764} C_VEL
LIN {X 0,Y 220.83,Z 259.466,A -85,B 0,C 180,E1 -20557.281,E2 -20557.281} C_VEL
LIN {X 0,Y 220.763,Z 259.476,A -85,B 0,C 180,E1 -20561.985,E2 -20561.985} C_VEL
LIN {X 0,Y 220.066,Z 259.571,A -85,B 0,C 180,E1 -20563.506,E2 -20563.506} C_VEL
LIN {X 0,Y 217.212,Z 259.922,A -85,B 0,C 180,E1 -20565.989,E2 -20565.989} C_VEL
LIN {X 0,Y 214.803,Z 260.225,A -85,B 0,C 180,E1 -20568.017,E2 -20568.017} C_VEL
LIN {X 0,Y 213.774,Z 260.356,A -85,B 0,C 180,E1 -20569.591,E2 -20569.591} C_VEL
LIN {X 0,Y 213.691,Z 260.363,A -85,B 0,C 180,E1 -20570.125,E2 -20570.125} C_VEL
LIN {X 0,Y 213.826,Z 260.43,A -85,B 0,C 180,E1 -20573.02,E2 -20573.02} C_VEL
LIN {X 0,Y 215.223,Z 267.035,A -85,B 0,C 180,E1 -20576.225,E2 -20576.225} C_VEL
LIN {X 0,Y 216.803,Z 271.218,A -85,B 0,C 180,E1 -20576.707,E2 -20576.707} C_VEL
LIN {X 0,Y 225.8,Z 295.871,A -85,B 0,C 180,E1 -20578.771,E2 -20578.771} C_VEL
LIN {X 0,Y 226.848,Z 302.034,A -85,B 0,C 180,E1 -20579.131,E2 -20579.131} C_VEL
LIN {X 0,Y 228.676,Z 316.017,A -85,B 0,C 180,E1 -20579.877,E2 -20579.877} C_VEL
LIN {X 0,Y 226.085,Z 374.313,A -85,B 0,C 180,E1 -20581.952,E2 -20581.952} C_VEL
LIN {X 0,Y 225.015,Z 387.863,A -85,B 0,C 180,E1 -20582.754,E2 -20582.754} C_VEL
LIN {X 0,Y 223.689,Z 399.763,A -85,B 0,C 180,E1 -20583.777,E2 -20583.777} C_VEL
LIN {X 0,Y 221.878,Z 411.984,A -85,B 0,C 180,E1 -20585.182,E2 -20585.182} C_VEL
LIN {X 0,Y 219.891,Z 423.62,A -85,B 0,C 180,E1 -20586.948,E2 -20586.948} C_VEL
LIN {X 0,Y 218.09,Z 434.186,A -85,B 0,C 180,E1 -20588.988,E2 -20588.988} C_VEL
LIN {X 0,Y 216.512,Z 442.826,A -85,B 0,C 180,E1 -20591.056,E2 -20591.056} C_VEL
LIN {X 0,Y 214.946,Z 450.759,A -85,B 0,C 180,E1 -20593.373,E2 -20593.373} C_VEL
LIN {X 0,Y 213.417,Z 458.481,A -85,B 0,C 180,E1 -20596.184,E2 -20596.184} C_VEL
LIN {X 0,Y 212.33,Z 465.611,A -85,B 0,C 180,E1 -20599.508,E2 -20599.508} C_VEL
LIN {X 0,Y 211.722,Z 470.282,A -85,B 0,C 180,E1 -20602.367,E2 -20602.367} C_VEL
LIN {X 0,Y 211.425,Z 474.402,A -85,B 0,C 180,E1 -20605.852,E2 -20605.852} C_VEL
LIN {X 0,Y 211.397,Z 476.278,A -85,B 0,C 180,E1 -20608.092,E2 -20608.092} C_VEL
LIN {X 0,Y 211.471,Z 477.37,A -85,B 0,C 180,E1 -20609.997,E2 -20609.997} C_VEL
LIN {X 0,Y 211.392,Z 478.04,A -85,B 0,C 180,E1 -20611.902,E2 -20611.902} C_VEL
LIN {X 0,Y 211.418,Z 478.339,A -85,B 0,C 180,E1 -20614.12,E2 -20614.12} C_VEL
LIN {X 0,Y 211.852,Z 477.665,A -85,B 0,C 180,E1 -20617.622,E2 -20617.622} C_VEL
LIN {X 0,Y 212.895,Z 475.397,A -85,B 0,C 180,E1 -20621.421,E2 -20621.421} C_VEL
LIN {X 0,Y 214.227,Z 472.611,A -85,B 0,C 180,E1 -20624.24,E2 -20624.24} C_VEL
LIN {X 0,Y 215.975,Z 468.825,A -85,B 0,C 180,E1 -20627.026,E2 -20627.026} C_VEL
LIN {X 0,Y 218.499,Z 463.924,A -85,B 0,C 180,E1 -20629.735,E2 -20629.735} C_VEL
LIN {X 0,Y 221.355,Z 457.792,A -85,B 0,C 180,E1 -20632.392,E2 -20632.392} C_VEL
LIN {X 0,Y 223.87,Z 451.626,A -85,B 0,C 180,E1 -20634.576,E2 -20634.576} C_VEL
LIN {X 0,Y 227.481,Z 442.642,A -85,B 0,C 180,E1 -20637.106,E2 -20637.106} C_VEL
LIN {X 0,Y 231.321,Z 432.326,A -85,B 0,C 180,E1 -20639.331,E2 -20639.331} C_VEL
LIN {X 0,Y 234.701,Z 421.935,A -85,B 0,C 180,E1 -20641.097,E2 -20641.097} C_VEL
LIN {X 0,Y 237.938,Z 410.45,A -85,B 0,C 180,E1 -20642.615,E2 -20642.615} C_VEL
LIN {X 0,Y 240.912,Z 397.363,A -85,B 0,C 180,E1 -20643.908,E2 -20643.908} C_VEL
LIN {X 0,Y 243.318,Z 384.043,A -85,B 0,C 180,E1 -20644.841,E2 -20644.841} C_VEL
LIN {X 0,Y 245.012,Z 369.884,A -85,B 0,C 180,E1 -20645.478,E2 -20645.478} C_VEL
LIN {X 0,Y 248.456,Z 321.975,A -85,B 0,C 180,E1 -20647.089,E2 -20647.089} C_VEL
LIN {X 0,Y 247.682,Z 319.311,A -85,B 0,C 180,E1 -20647.425,E2 -20647.425} C_VEL
LIN {X 0,Y 243.028,Z 308.223,A -85,B 0,C 180,E1 -20649.295,E2 -20649.295} C_VEL
LIN {X 0,Y 237.927,Z 298.08,A -85,B 0,C 180,E1 -20651.472,E2 -20651.472} C_VEL
LIN {X 0,Y 233.916,Z 291.276,A -85,B 0,C 180,E1 -20653.315,E2 -20653.315} C_VEL
LIN {X 0,Y 231.338,Z 287.051,A -85,B 0,C 180,E1 -20654.589,E2 -20654.589} C_VEL
LIN {X 0,Y 228.064,Z 282.006,A -85,B 0,C 180,E1 -20656.34,E2 -20656.34} C_VEL
LIN {X 0,Y 224.537,Z 276.864,A -85,B 0,C 180,E1 -20658.435,E2 -20658.435} C_VEL
LIN {X 0,Y 221.36,Z 272.608,A -85,B 0,C 180,E1 -20660.569,E2 -20660.569} C_VEL
LIN {X 0,Y 220.152,Z 270.836,A -85,B 0,C 180,E1 -20661.489,E2 -20661.489} C_VEL
LIN {X 0,Y 215.217,Z 264.456,A -85,B 0,C 180,E1 -20666.083,E2 -20666.083} C_VEL
LIN {X 0,Y 214.622,Z 262.932,A -85,B 0,C 180,E1 -20668.391,E2 -20668.391} C_VEL
LIN {X 0,Y 213.931,Z 261.114,A -85,B 0,C 180,E1 -20672.606,E2 -20672.606} C_VEL
LIN {X 0,Y 213.781,Z 260.392,A -85,B 0,C 180,E1 -20676.24,E2 -20676.24} C_VEL
LIN {X 0,Y 213.792,Z 260.362,A -85,B 0,C 180,E1 -20680.797,E2 -20680.797} C_VEL
LIN {X 0,Y 213.935,Z 260.556,A -85,B 0,C 180,E1 -20683.774,E2 -20683.774} C_VEL
LIN {X 0,Y 214.799,Z 262.741,A -85,B 0,C 180,E1 -20689.455,E2 -20689.455} C_VEL
LIN {X 0,Y 216.364,Z 264.785,A -85,B 0,C 180,E1 -20691.348,E2 -20691.348} C_VEL
LIN {X 0,Y 220.628,Z 269.687,A -85,B 0,C 180,E1 -20694.963,E2 -20694.963} C_VEL
LIN {X 0,Y 223.119,Z 272.91,A -85,B 0,C 180,E1 -20696.724,E2 -20696.724} C_VEL
LIN {X 0,Y 225.1,Z 274.931,A -85,B 0,C 180,E1 -20697.953,E2 -20697.953} C_VEL
LIN {X 0,Y 228.929,Z 280.52,A -85,B 0,C 180,E1 -20700.197,E2 -20700.197} C_VEL
LIN {X 0,Y 235.449,Z 290.546,A -85,B 0,C 180,E1 -20703.465,E2 -20703.465} C_VEL
LIN {X 0,Y 239.536,Z 297.655,A -85,B 0,C 180,E1 -20705.286,E2 -20705.286} C_VEL
LIN {X 0,Y 245.129,Z 309.011,A -85,B 0,C 180,E1 -20707.615,E2 -20707.615} C_VEL
LIN {X 0,Y 248.726,Z 317.48,A -85,B 0,C 180,E1 -20709.013,E2 -20709.013} C_VEL
LIN {X 0,Y 244.727,Z 370.391,A -85,B 0,C 180,E1 -20710.801,E2 -20710.801} C_VEL
LIN {X 0,Y 242.96,Z 383.295,A -85,B 0,C 180,E1 -20711.492,E2 -20711.492} C_VEL
LIN {X 0,Y 240.569,Z 396.384,A -85,B 0,C 180,E1 -20712.537,E2 -20712.537} C_VEL
LIN {X 0,Y 237.682,Z 408.68,A -85,B 0,C 180,E1 -20713.889,E2 -20713.889} C_VEL
LIN {X 0,Y 234.584,Z 419.441,A -85,B 0,C 180,E1 -20715.407,E2 -20715.407} C_VEL
LIN {X 0,Y 231.233,Z 429.564,A -85,B 0,C 180,E1 -20717.224,E2 -20717.224} C_VEL
LIN {X 0,Y 227.594,Z 439.258,A -85,B 0,C 180,E1 -20719.454,E2 -20719.454} C_VEL
LIN {X 0,Y 223.763,Z 448.37,A -85,B 0,C 180,E1 -20722.127,E2 -20722.127} C_VEL
LIN {X 0,Y 220.58,Z 455.425,A -85,B 0,C 180,E1 -20724.83,E2 -20724.83} C_VEL
LIN {X 0,Y 217.651,Z 461.456,A -85,B 0,C 180,E1 -20727.813,E2 -20727.813} C_VEL
LIN {X 0,Y 215.722,Z 465.328,A -85,B 0,C 180,E1 -20730.313,E2 -20730.313} C_VEL
LIN {X 0,Y 213.544,Z 469.428,A -85,B 0,C 180,E1 -20734.003,E2 -20734.003} C_VEL
LIN {X 0,Y 212.193,Z 471.666,A -85,B 0,C 180,E1 -20737.361,E2 -20737.361} C_VEL
LIN {X 0,Y 211.504,Z 472.56,A -85,B 0,C 180,E1 -20740.165,E2 -20740.165} C_VEL
LIN {X 0,Y 211.112,Z 472.574,A -85,B 0,C 180,E1 -20742.919,E2 -20742.919} C_VEL
LIN {X 0,Y 210.954,Z 471.785,A -85,B 0,C 180,E1 -20745.609,E2 -20745.609} C_VEL
LIN {X 0,Y 210.944,Z 470.253,A -85,B 0,C 180,E1 -20748.22,E2 -20748.22} C_VEL
LIN {X 0,Y 211.429,Z 466.716,A -85,B 0,C 180,E1 -20751.89,E2 -20751.89} C_VEL
LIN {X 0,Y 212.102,Z 462.125,A -85,B 0,C 180,E1 -20755.144,E2 -20755.144} C_VEL
LIN {X 0,Y 213.02,Z 456.451,A -85,B 0,C 180,E1 -20758.142,E2 -20758.142} C_VEL
LIN {X 0,Y 214.408,Z 448.697,A -85,B 0,C 180,E1 -20761.321,E2 -20761.321} C_VEL
LIN {X 0,Y 215.98,Z 440.564,A -85,B 0,C 180,E1 -20763.945,E2 -20763.945} C_VEL
LIN {X 0,Y 217.853,Z 430.692,A -85,B 0,C 180,E1 -20766.474,E2 -20766.474} C_VEL
LIN {X 0,Y 219.773,Z 420.482,A -85,B 0,C 180,E1 -20768.562,E2 -20768.562} C_VEL
LIN {X 0,Y 221.679,Z 408.775,A -85,B 0,C 180,E1 -20770.446,E2 -20770.446} C_VEL
LIN {X 0,Y 223.515,Z 395.9,A -85,B 0,C 180,E1 -20772.033,E2 -20772.033} C_VEL
LIN {X 0,Y 224.953,Z 382.459,A -85,B 0,C 180,E1 -20773.235,E2 -20773.235} C_VEL
LIN {X 0,Y 226.084,Z 369.12,A -85,B 0,C 180,E1 -20774.038,E2 -20774.038} C_VEL
LIN {X 0,Y 229.02,Z 304.561,A -85,B 0,C 180,E1 -20776.339,E2 -20776.339} C_VEL
LIN {X 0,Y 228.107,Z 299.463,A -85,B 0,C 180,E1 -20776.637,E2 -20776.637} C_VEL
LIN {X 0,Y 219.914,Z 276.267,A -85,B 0,C 180,E1 -20778.503,E2 -20778.503} C_VEL
LIN {X 0,Y 214.422,Z 262.074,A -85,B 0,C 180,E1 -20779.826,E2 -20779.826} C_VEL
LIN {X 0,Y 214.175,Z 260.682,A -85,B 0,C 180,E1 -20780.343,E2 -20780.343} C_VEL
LIN {X 0,Y 214.121,Z 260.315,A -85,B 0,C 180,E1 -20781.034,E2 -20781.034} C_VEL
LIN {X 0,Y 214.044,Z 260.324,A -85,B 0,C 180,E1 -20784.35,E2 -20784.35} C_VEL
LIN {X 0,Y 214.417,Z 260.277,A -85,B 0,C 180,E1 -20788.125,E2 -20788.125} C_VEL
LIN {X 0,Y 214.418,Z 260.276,A -85,B 0,C 180,E1 -20791.882,E2 -20791.882} C_VEL
LIN {X 0,Y 214.16,Z 260.308,A -85,B 0,C 180,E1 -20797.546,E2 -20797.546} C_VEL
LIN {X 0,Y 213.95,Z 260.323,A -85,B 0,C 180,E1 -20801.37,E2 -20801.37} C_VEL
LIN {X 0,Y 213.861,Z 260.344,A -85,B 0,C 180,E1 -20805.245,E2 -20805.245} C_VEL
LIN {X 0,Y 213.779,Z 260.338,A -85,B 0,C 180,E1 -20809.196,E2 -20809.196} C_VEL
LIN {X 0,Y 213.76,Z 260.358,A -85,B 0,C 180,E1 -20813.24,E2 -20813.24} C_VEL
LIN {X 0,Y 213.782,Z 260.332,A -85,B 0,C 180,E1 -20817.46,E2 -20817.46} C_VEL
LIN {X 0,Y 213.725,Z 260.35,A -85,B 0,C 180,E1 -20821.748,E2 -20821.748} C_VEL
LIN {X 0,Y 213.712,Z 260.363,A -85,B 0,C 180,E1 -20826.298,E2 -20826.298} C_VEL
LIN {X 0,Y 213.76,Z 260.356,A -85,B 0,C 180,E1 -20831.118,E2 -20831.118} C_VEL
LIN {X 0,Y 213.803,Z 260.351,A -85,B 0,C 180,E1 -20833.705,E2 -20833.705} C_VEL
LIN {X 0,Y 213.809,Z 260.343,A -85,B 0,C 180,E1 -20836.369,E2 -20836.369} C_VEL
LIN {X 0,Y 213.797,Z 260.352,A -85,B 0,C 180,E1 -20839.122,E2 -20839.122} C_VEL
LIN {X 0,Y 213.735,Z 260.354,A -85,B 0,C 180,E1 -20843.728,E2 -20843.728} C_VEL
LIN {X 0,Y 213.75,Z 260.356,A -85,B 0,C 180,E1 -20848.277,E2 -20848.277} C_VEL
LIN {X 0,Y 213.811,Z 260.348,A -85,B 0,C 180,E1 -20852.617,E2 -20852.617} C_VEL
LIN {X 0,Y 213.806,Z 260.347,A -85,B 0,C 180,E1 -20856.989,E2 -20856.989} C_VEL
LIN {X 0,Y 213.878,Z 260.336,A -85,B 0,C 180,E1 -20862.812,E2 -20862.812} C_VEL
LIN {X 0,Y 213.937,Z 260.331,A -85,B 0,C 180,E1 -20866.719,E2 -20866.719} C_VEL
LIN {X 0,Y 214.135,Z 260.306,A -85,B 0,C 180,E1 -20870.568,E2 -20870.568} C_VEL
LIN {X 0,Y 214.082,Z 260.313,A -85,B 0,C 180,E1 -20874.361,E2 -20874.361} C_VEL
LIN {X 0,Y 214.415,Z 260.276,A -85,B 0,C 180,E1 -20878.134,E2 -20878.134} C_VEL
LIN {X 0,Y 214.52,Z 260.258,A -85,B 0,C 180,E1 -20880.012,E2 -20880.012} C_VEL
LIN {X 0,Y 214.414,Z 260.26,A -85,B 0,C 180,E1 -20881.891,E2 -20881.891} C_VEL
LIN {X 0,Y 214.191,Z 260.282,A -85,B 0,C 180,E1 -20887.554,E2 -20887.554} C_VEL
LIN {X 0,Y 214.009,Z 260.325,A -85,B 0,C 180,E1 -20891.376,E2 -20891.376} C_VEL
LIN {X 0,Y 213.916,Z 260.331,A -85,B 0,C 180,E1 -20895.25,E2 -20895.25} C_VEL
LIN {X 0,Y 213.815,Z 260.326,A -85,B 0,C 180,E1 -20899.201,E2 -20899.201} C_VEL
LIN {X 0,Y 213.818,Z 260.351,A -85,B 0,C 180,E1 -20903.242,E2 -20903.242} C_VEL
LIN {X 0,Y 213.811,Z 260.338,A -85,B 0,C 180,E1 -20907.435,E2 -20907.435} C_VEL
LIN {X 0,Y 213.786,Z 260.354,A -85,B 0,C 180,E1 -20911.747,E2 -20911.747} C_VEL
LIN {X 0,Y 213.77,Z 260.341,A -85,B 0,C 180,E1 -20916.295,E2 -20916.295} C_VEL
LIN {X 0,Y 213.721,Z 260.357,A -85,B 0,C 180,E1 -20921.136,E2 -20921.136} C_VEL
LIN {X 0,Y 213.711,Z 260.361,A -85,B 0,C 180,E1 -20923.691,E2 -20923.691} C_VEL
LIN {X 0,Y 213.711,Z 260.357,A -85,B 0,C 180,E1 -20926.356,E2 -20926.356} C_VEL
LIN {X 0,Y 213.691,Z 260.363,A -85,B 0,C 180,E1 -20930.125,E2 -20930.125} C_VEL
LIN {X 0,Y 213.042,Z 260.476,A -85,B 0,C 180,E1 -20931.282,E2 -20931.282} C_VEL
LIN {X 0,Y 211.565,Z 260.918,A -85,B 0,C 180,E1 -20932.396,E2 -20932.396} C_VEL
LIN {X 0,Y 210.272,Z 261.679,A -85,B 0,C 180,E1 -20933.212,E2 -20933.212} C_VEL
LIN {X 0,Y 208.071,Z 266.033,A -85,B 0,C 180,E1 -20934.947,E2 -20934.947} C_VEL
LIN {X 0,Y 208.069,Z 267.323,A -85,B 0,C 180,E1 -20935.379,E2 -20935.379} C_VEL
LIN {X 0,Y 216.017,Z 288.167,A -85,B 0,C 180,E1 -20937.335,E2 -20937.335} C_VEL
LIN {X 0,Y 219.897,Z 299.732,A -85,B 0,C 180,E1 -20938.277,E2 -20938.277} C_VEL
LIN {X 0,Y 222.076,Z 317.6,A -85,B 0,C 180,E1 -20939.255,E2 -20939.255} C_VEL
LIN {X 0,Y 219.385,Z 374.606,A -85,B 0,C 180,E1 -20941.343,E2 -20941.343} C_VEL
LIN {X 0,Y 218.293,Z 388.009,A -85,B 0,C 180,E1 -20942.168,E2 -20942.168} C_VEL
LIN {X 0,Y 216.88,Z 400.407,A -85,B 0,C 180,E1 -20943.278,E2 -20943.278} C_VEL
LIN {X 0,Y 215.136,Z 411.613,A -85,B 0,C 180,E1 -20944.608,E2 -20944.608} C_VEL
LIN {X 0,Y 213.089,Z 423.305,A -85,B 0,C 180,E1 -20946.425,E2 -20946.425} C_VEL
LIN {X 0,Y 211.221,Z 433.909,A -85,B 0,C 180,E1 -20948.527,E2 -20948.527} C_VEL
LIN {X 0,Y 209.742,Z 441.671,A -85,B 0,C 180,E1 -20950.42,E2 -20950.42} C_VEL
LIN {X 0,Y 208.084,Z 449.799,A -85,B 0,C 180,E1 -20952.807,E2 -20952.807} C_VEL
LIN {X 0,Y 206.711,Z 456.518,A -85,B 0,C 180,E1 -20955.224,E2 -20955.224} C_VEL
LIN {X 0,Y 205.592,Z 463.121,A -85,B 0,C 180,E1 -20958.161,E2 -20958.161} C_VEL
LIN {X 0,Y 204.846,Z 468.319,A -85,B 0,C 180,E1 -20961.115,E2 -20961.115} C_VEL
LIN {X 0,Y 204.436,Z 472.318,A -85,B 0,C 180,E1 -20964.077,E2 -20964.077} C_VEL
LIN {X 0,Y 204.329,Z 474.36,A -85,B 0,C 180,E1 -20966.052,E2 -20966.052} C_VEL
LIN {X 0,Y 204.305,Z 475.97,A -85,B 0,C 180,E1 -20968.025,E2 -20968.025} C_VEL
LIN {X 0,Y 204.375,Z 477.15,A -85,B 0,C 180,E1 -20969.997,E2 -20969.997} C_VEL
LIN {X 0,Y 204.288,Z 478.18,A -85,B 0,C 180,E1 -20973.78,E2 -20973.78} C_VEL
LIN {X 0,Y 204.449,Z 478.13,A -85,B 0,C 180,E1 -20975.916,E2 -20975.916} C_VEL
LIN {X 0,Y 204.791,Z 477.681,A -85,B 0,C 180,E1 -20977.886,E2 -20977.886} C_VEL
LIN {X 0,Y 205.924,Z 475.524,A -85,B 0,C 180,E1 -20981.813,E2 -20981.813} C_VEL
LIN {X 0,Y 207.325,Z 472.843,A -85,B 0,C 180,E1 -20984.725,E2 -20984.725} C_VEL
LIN {X 0,Y 209.211,Z 469.171,A -85,B 0,C 180,E1 -20987.594,E2 -20987.594} C_VEL
LIN {X 0,Y 211.85,Z 464.417,A -85,B 0,C 180,E1 -20990.381,E2 -20990.381} C_VEL
LIN {X 0,Y 215.317,Z 457.368,A -85,B 0,C 180,E1 -20993.554,E2 -20993.554} C_VEL
LIN {X 0,Y 218.106,Z 451.094,A -85,B 0,C 180,E1 -20995.782,E2 -20995.782} C_VEL
LIN {X 0,Y 221.262,Z 443.632,A -85,B 0,C 180,E1 -20997.934,E2 -20997.934} C_VEL
LIN {X 0,Y 224.847,Z 434.64,A -85,B 0,C 180,E1 -21000.003,E2 -21000.003} C_VEL
LIN {X 0,Y 228.763,Z 423.587,A -85,B 0,C 180,E1 -21001.998,E2 -21001.998} C_VEL
LIN {X 0,Y 232.094,Z 412.6,A -85,B 0,C 180,E1 -21003.543,E2 -21003.543} C_VEL
LIN {X 0,Y 235.211,Z 400.411,A -85,B 0,C 180,E1 -21004.847,E2 -21004.847} C_VEL
LIN {X 0,Y 237.803,Z 387.489,A -85,B 0,C 180,E1 -21005.837,E2 -21005.837} C_VEL
LIN {X 0,Y 239.739,Z 374.078,A -85,B 0,C 180,E1 -21006.538,E2 -21006.538} C_VEL
LIN {X 0,Y 243.616,Z 323.886,A -85,B 0,C 180,E1 -21008.256,E2 -21008.256} C_VEL
LIN {X 0,Y 238.975,Z 312.502,A -85,B 0,C 180,E1 -21010.263,E2 -21010.263} C_VEL
LIN {X 0,Y 234.197,Z 302.704,A -85,B 0,C 180,E1 -21012.443,E2 -21012.443} C_VEL
LIN {X 0,Y 229.044,Z 293.633,A -85,B 0,C 180,E1 -21015.032,E2 -21015.032} C_VEL
LIN {X 0,Y 225.391,Z 287.935,A -85,B 0,C 180,E1 -21017.093,E2 -21017.093} C_VEL
LIN {X 0,Y 222.088,Z 282.964,A -85,B 0,C 180,E1 -21019.169,E2 -21019.169} C_VEL
LIN {X 0,Y 219.001,Z 278.485,A -85,B 0,C 180,E1 -21021.405,E2 -21021.405} C_VEL
LIN {X 0,Y 217.638,Z 276.765,A -85,B 0,C 180,E1 -21022.491,E2 -21022.491} C_VEL
LIN {X 0,Y 212.987,Z 270.496,A -85,B 0,C 180,E1 -21027.141,E2 -21027.141} C_VEL
LIN {X 0,Y 209.191,Z 266.121,A -85,B 0,C 180,E1 -21033.898,E2 -21033.898} C_VEL
LIN {X 0,Y 208.624,Z 265.227,A -85,B 0,C 180,E1 -21037.03,E2 -21037.03} C_VEL
LIN {X 0,Y 209.08,Z 265.611,A -85,B 0,C 180,E1 -21041.872,E2 -21041.872} C_VEL
LIN {X 0,Y 210.656,Z 267.391,A -85,B 0,C 180,E1 -21045.67,E2 -21045.67} C_VEL
LIN {X 0,Y 213.676,Z 270.089,A -85,B 0,C 180,E1 -21049.734,E2 -21049.734} C_VEL
LIN {X 0,Y 218.543,Z 276.019,A -85,B 0,C 180,E1 -21054.305,E2 -21054.305} C_VEL
LIN {X 0,Y 221.3,Z 279.627,A -85,B 0,C 180,E1 -21056.347,E2 -21056.347} C_VEL
LIN {X 0,Y 222.807,Z 281.245,A -85,B 0,C 180,E1 -21057.328,E2 -21057.328} C_VEL
LIN {X 0,Y 226.313,Z 286.503,A -85,B 0,C 180,E1 -21059.488,E2 -21059.488} C_VEL
LIN {X 0,Y 230.933,Z 293.983,A -85,B 0,C 180,E1 -21062.012,E2 -21062.012} C_VEL
LIN {X 0,Y 234.445,Z 299.818,A -85,B 0,C 180,E1 -21063.722,E2 -21063.722} C_VEL
LIN {X 0,Y 239.723,Z 310.29,A -85,B 0,C 180,E1 -21066.1,E2 -21066.1} C_VEL
LIN {X 0,Y 243.754,Z 319.783,A -85,B 0,C 180,E1 -21067.828,E2 -21067.828} C_VEL
LIN {X 0,Y 239.768,Z 371.035,A -85,B 0,C 180,E1 -21069.607,E2 -21069.607} C_VEL
LIN {X 0,Y 237.866,Z 384.297,A -85,B 0,C 180,E1 -21070.342,E2 -21070.342} C_VEL
LIN {X 0,Y 235.493,Z 396.617,A -85,B 0,C 180,E1 -21071.348,E2 -21071.348} C_VEL
LIN {X 0,Y 232.791,Z 407.619,A -85,B 0,C 180,E1 -21072.554,E2 -21072.554} C_VEL
LIN {X 0,Y 229.301,Z 419.173,A -85,B 0,C 180,E1 -21074.181,E2 -21074.181} C_VEL
LIN {X 0,Y 225.981,Z 428.771,A -85,B 0,C 180,E1 -21075.914,E2 -21075.914} C_VEL
LIN {X 0,Y 222.717,Z 437.239,A -85,B 0,C 180,E1 -21077.81,E2 -21077.81} C_VEL
LIN {X 0,Y 219.093,Z 445.649,A -85,B 0,C 180,E1 -21080.157,E2 -21080.157} C_VEL
LIN {X 0,Y 215.282,Z 453.683,A -85,B 0,C 180,E1 -21083.048,E2 -21083.048} C_VEL
LIN {X 0,Y 212.659,Z 458.869,A -85,B 0,C 180,E1 -21085.428,E2 -21085.428} C_VEL
LIN {X 0,Y 210.404,Z 463.125,A -85,B 0,C 180,E1 -21087.864,E2 -21087.864} C_VEL
LIN {X 0,Y 208.506,Z 466.55,A -85,B 0,C 180,E1 -21090.354,E2 -21090.354} C_VEL
LIN {X 0,Y 206.996,Z 469.166,A -85,B 0,C 180,E1 -21092.887,E2 -21092.887} C_VEL
LIN {X 0,Y 205.74,Z 471.091,A -85,B 0,C 180,E1 -21095.482,E2 -21095.482} C_VEL
LIN {X 0,Y 204.869,Z 472.305,A -85,B 0,C 180,E1 -21098.113,E2 -21098.113} C_VEL
LIN {X 0,Y 204.307,Z 472.759,A -85,B 0,C 180,E1 -21100.825,E2 -21100.825} C_VEL
LIN {X 0,Y 203.94,Z 472.449,A -85,B 0,C 180,E1 -21103.646,E2 -21103.646} C_VEL
LIN {X 0,Y 203.826,Z 471.363,A -85,B 0,C 180,E1 -21106.406,E2 -21106.406} C_VEL
LIN {X 0,Y 203.944,Z 469.378,A -85,B 0,C 180,E1 -21109.275,E2 -21109.275} C_VEL
LIN {X 0,Y 204.389,Z 466.332,A -85,B 0,C 180,E1 -21112.24,E2 -21112.24} C_VEL
LIN {X 0,Y 205.031,Z 461.984,A -85,B 0,C 180,E1 -21115.324,E2 -21115.324} C_VEL
LIN {X 0,Y 206.027,Z 456.109,A -85,B 0,C 180,E1 -21118.487,E2 -21118.487} C_VEL
LIN {X 0,Y 207.447,Z 448.411,A -85,B 0,C 180,E1 -21121.709,E2 -21121.709} C_VEL
LIN {X 0,Y 209.204,Z 439.668,A -85,B 0,C 180,E1 -21124.556,E2 -21124.556} C_VEL
LIN {X 0,Y 210.899,Z 430.906,A -85,B 0,C 180,E1 -21126.853,E2 -21126.853} C_VEL
LIN {X 0,Y 212.825,Z 420.962,A -85,B 0,C 180,E1 -21128.958,E2 -21128.958} C_VEL
LIN {X 0,Y 214.797,Z 409.331,A -85,B 0,C 180,E1 -21130.905,E2 -21130.905} C_VEL
LIN {X 0,Y 216.687,Z 396.512,A -85,B 0,C 180,E1 -21132.545,E2 -21132.545} C_VEL
LIN {X 0,Y 218.171,Z 383.463,A -85,B 0,C 180,E1 -21133.77,E2 -21133.77} C_VEL
LIN {X 0,Y 219.42,Z 369.295,A -85,B 0,C 180,E1 -21134.66,E2 -21134.66} C_VEL
LIN {X 0,Y 222.432,Z 304.958,A -85,B 0,C 180,E1 -21137.022,E2 -21137.022} C_VEL
LIN {X 0,Y 221.304,Z 300.228,A -85,B 0,C 180,E1 -21137.343,E2 -21137.343} C_VEL
LIN {X 0,Y 213.549,Z 278.33,A -85,B 0,C 180,E1 -21139.187,E2 -21139.187} C_VEL
LIN {X 0,Y 207.358,Z 262.438,A -85,B 0,C 180,E1 -21140.739,E2 -21140.739} C_VEL
LIN {X 0,Y 207.104,Z 261.384,A -85,B 0,C 180,E1 -21141.097,E2 -21141.097} C_VEL
LIN {X 0,Y 207.005,Z 261.201,A -85,B 0,C 180,E1 -21144.158,E2 -21144.158} C_VEL
LIN {X 0,Y 207.35,Z 261.157,A -85,B 0,C 180,E1 -21148.061,E2 -21148.061} C_VEL
LIN {X 0,Y 207.454,Z 261.136,A -85,B 0,C 180,E1 -21150.003,E2 -21150.003} C_VEL
LIN {X 0,Y 207.35,Z 261.156,A -85,B 0,C 180,E1 -21151.946,E2 -21151.946} C_VEL
LIN {X 0,Y 207.101,Z 261.186,A -85,B 0,C 180,E1 -21157.805,E2 -21157.805} C_VEL
LIN {X 0,Y 207.036,Z 261.179,A -85,B 0,C 180,E1 -21160.219,E2 -21160.219} C_VEL
LIN {X 0,Y 206.797,Z 261.219,A -85,B 0,C 180,E1 -21165.779,E2 -21165.779} C_VEL
LIN {X 0,Y 206.707,Z 261.223,A -85,B 0,C 180,E1 -21169.88,E2 -21169.88} C_VEL
LIN {X 0,Y 206.697,Z 261.236,A -85,B 0,C 180,E1 -21174.084,E2 -21174.084} C_VEL
LIN {X 0,Y 206.69,Z 261.206,A -85,B 0,C 180,E1 -21178.43,E2 -21178.43} C_VEL
LIN {X 0,Y 206.662,Z 261.238,A -85,B 0,C 180,E1 -21182.968,E2 -21182.968} C_VEL
LIN {X 0,Y 206.686,Z 261.235,A -85,B 0,C 180,E1 -21187.742,E2 -21187.742} C_VEL
LIN {X 0,Y 206.689,Z 261.236,A -85,B 0,C 180,E1 -21191.601,E2 -21191.601} C_VEL
LIN {X 0,Y 206.714,Z 261.228,A -85,B 0,C 180,E1 -21195.563,E2 -21195.563} C_VEL
LIN {X 0,Y 206.72,Z 261.232,A -85,B 0,C 180,E1 -21199.783,E2 -21199.783} C_VEL
LIN {X 0,Y 206.717,Z 261.234,A -85,B 0,C 180,E1 -21202.287,E2 -21202.287} C_VEL
LIN {X 0,Y 206.684,Z 261.233,A -85,B 0,C 180,E1 -21207.058,E2 -21207.058} C_VEL
LIN {X 0,Y 206.748,Z 261.227,A -85,B 0,C 180,E1 -21212.112,E2 -21212.112} C_VEL
LIN {X 0,Y 206.741,Z 261.225,A -85,B 0,C 180,E1 -21216.62,E2 -21216.62} C_VEL
LIN {X 0,Y 206.815,Z 261.215,A -85,B 0,C 180,E1 -21222.206,E2 -21222.206} C_VEL
LIN {X 0,Y 206.876,Z 261.211,A -85,B 0,C 180,E1 -21226.257,E2 -21226.257} C_VEL
LIN {X 0,Y 207.079,Z 261.186,A -85,B 0,C 180,E1 -21230.244,E2 -21230.244} C_VEL
LIN {X 0,Y 207.045,Z 261.186,A -85,B 0,C 180,E1 -21234.169,E2 -21234.169} C_VEL
LIN {X 0,Y 207.355,Z 261.156,A -85,B 0,C 180,E1 -21238.071,E2 -21238.071} C_VEL
LIN {X 0,Y 207.488,Z 261.133,A -85,B 0,C 180,E1 -21240.013,E2 -21240.013} C_VEL
LIN {X 0,Y 207.354,Z 261.138,A -85,B 0,C 180,E1 -21241.955,E2 -21241.955} C_VEL
LIN {X 0,Y 207.136,Z 261.161,A -85,B 0,C 180,E1 -21247.812,E2 -21247.812} C_VEL
LIN {X 0,Y 206.932,Z 261.207,A -85,B 0,C 180,E1 -21251.77,E2 -21251.77} C_VEL
LIN {X 0,Y 206.844,Z 261.211,A -85,B 0,C 180,E1 -21255.785,E2 -21255.785} C_VEL
LIN {X 0,Y 206.736,Z 261.211,A -85,B 0,C 180,E1 -21259.886,E2 -21259.886} C_VEL
LIN {X 0,Y 206.759,Z 261.229,A -85,B 0,C 180,E1 -21264.085,E2 -21264.085} C_VEL
LIN {X 0,Y 206.713,Z 261.217,A -85,B 0,C 180,E1 -21268.436,E2 -21268.436} C_VEL
LIN {X 0,Y 206.722,Z 261.236,A -85,B 0,C 180,E1 -21272.966,E2 -21272.966} C_VEL
LIN {X 0,Y 206.729,Z 261.222,A -85,B 0,C 180,E1 -21275.318,E2 -21275.318} C_VEL
LIN {X 0,Y 206.672,Z 261.239,A -85,B 0,C 180,E1 -21280.262,E2 -21280.262} C_VEL
LIN {X 0,Y 206.643,Z 261.241,A -85,B 0,C 180,E1 -21285.593,E2 -21285.593} C_VEL
LIN {X 0,Y 206.663,Z 261.239,A -85,B 0,C 180,E1 -21290.117,E2 -21290.117} C_VEL
LIN {X 0,Y 206.78,Z 261.422,A -85,B 0,C 180,E1 -21292.559,E2 -21292.559} C_VEL
LIN {X 0,Y 208.013,Z 267.06,A -85,B 0,C 180,E1 -21295.331,E2 -21295.331} C_VEL
LIN {X 0,Y 208.069,Z 267.323,A -85,B 0,C 180,E1 -21295.379,E2 -21295.379} C_VEL
LIN {X 0,Y 209.856,Z 274.667,A -85,B 0,C 180,E1 -21295.971,E2 -21295.971} C_VEL
LIN {X 0,Y 211.576,Z 294.066,A -85,B 0,C 180,E1 -21297.035,E2 -21297.035} C_VEL
LIN {X 0,Y 212.334,Z 297.831,A -85,B 0,C 180,E1 -21297.303,E2 -21297.303} C_VEL
LIN {X 0,Y 213.647,Z 302.456,A -85,B 0,C 180,E1 -21297.663,E2 -21297.663} C_VEL
LIN {X 0,Y 215.507,Z 318.003,A -85,B 0,C 180,E1 -21298.545,E2 -21298.545} C_VEL
LIN {X 0,Y 212.719,Z 374.877,A -85,B 0,C 180,E1 -21300.696,E2 -21300.696} C_VEL
LIN {X 0,Y 211.509,Z 388.874,A -85,B 0,C 180,E1 -21301.6,E2 -21301.6} C_VEL
LIN {X 0,Y 210.076,Z 401.039,A -85,B 0,C 180,E1 -21302.745,E2 -21302.745} C_VEL
LIN {X 0,Y 208.105,Z 412.823,A -85,B 0,C 180,E1 -21304.224,E2 -21304.224} C_VEL
LIN {X 0,Y 206.073,Z 424.295,A -85,B 0,C 180,E1 -21306.106,E2 -21306.106} C_VEL
LIN {X 0,Y 204.206,Z 434.381,A -85,B 0,C 180,E1 -21308.201,E2 -21308.201} C_VEL
LIN {X 0,Y 202.301,Z 444.035,A -85,B 0,C 180,E1 -21310.726,E2 -21310.726} C_VEL
LIN {X 0,Y 200.404,Z 453.099,A -85,B 0,C 180,E1 -21313.703,E2 -21313.703} C_VEL
LIN {X 0,Y 198.947,Z 460.35,A -85,B 0,C 180,E1 -21316.722,E2 -21316.722} C_VEL
LIN {X 0,Y 198.05,Z 466.11,A -85,B 0,C 180,E1 -21319.777,E2 -21319.777} C_VEL
LIN {X 0,Y 197.467,Z 470.606,A -85,B 0,C 180,E1 -21322.841,E2 -21322.841} C_VEL
LIN {X 0,Y 197.214,Z 474.377,A -85,B 0,C 180,E1 -21326.363,E2 -21326.363} C_VEL
LIN {X 0,Y 197.28,Z 476.878,A -85,B 0,C 180,E1 -21329.997,E2 -21329.997} C_VEL
LIN {X 0,Y 197.198,Z 478.024,A -85,B 0,C 180,E1 -21333.565,E2 -21333.565} C_VEL
LIN {X 0,Y 197.389,Z 478.054,A -85,B 0,C 180,E1 -21336.128,E2 -21336.128} C_VEL
LIN {X 0,Y 197.746,Z 477.66,A -85,B 0,C 180,E1 -21338.169,E2 -21338.169} C_VEL
LIN {X 0,Y 198.255,Z 476.874,A -85,B 0,C 180,E1 -21340.206,E2 -21340.206} C_VEL
LIN {X 0,Y 199.911,Z 474.043,A -85,B 0,C 180,E1 -21344.242,E2 -21344.242} C_VEL
LIN {X 0,Y 201.739,Z 470.835,A -85,B 0,C 180,E1 -21347.221,E2 -21347.221} C_VEL
LIN {X 0,Y 204.243,Z 466.584,A -85,B 0,C 180,E1 -21350.123,E2 -21350.123} C_VEL
LIN {X 0,Y 207.837,Z 460.169,A -85,B 0,C 180,E1 -21353.407,E2 -21353.407} C_VEL
LIN {X 0,Y 211.167,Z 453.247,A -85,B 0,C 180,E1 -21356.162,E2 -21356.162} C_VEL
LIN {X 0,Y 215.087,Z 444.687,A -85,B 0,C 180,E1 -21358.809,E2 -21358.809} C_VEL
LIN {X 0,Y 218.813,Z 435.975,A -85,B 0,C 180,E1 -21360.92,E2 -21360.92} C_VEL
LIN {X 0,Y 222.892,Z 425.337,A -85,B 0,C 180,E1 -21362.946,E2 -21362.946} C_VEL
LIN {X 0,Y 226.305,Z 414.784,A -85,B 0,C 180,E1 -21364.52,E2 -21364.52} C_VEL
LIN {X 0,Y 229.517,Z 403.165,A -85,B 0,C 180,E1 -21365.843,E2 -21365.843} C_VEL
LIN {X 0,Y 232.456,Z 390.119,A -85,B 0,C 180,E1 -21366.93,E2 -21366.93} C_VEL
LIN {X 0,Y 234.609,Z 376.83,A -85,B 0,C 180,E1 -21367.683,E2 -21367.683} C_VEL
LIN {X 0,Y 236.53,Z 354.894,A -85,B 0,C 180,E1 -21368.512,E2 -21368.512} C_VEL
LIN {X 0,Y 238.869,Z 326.824,A -85,B 0,C 180,E1 -21369.453,E2 -21369.453} C_VEL
LIN {X 0,Y 237.521,Z 322.812,A -85,B 0,C 180,E1 -21370.099,E2 -21370.099} C_VEL
LIN {X 0,Y 233.703,Z 313.882,A -85,B 0,C 180,E1 -21371.881,E2 -21371.881} C_VEL
LIN {X 0,Y 230.157,Z 306.676,A -85,B 0,C 180,E1 -21373.661,E2 -21373.661} C_VEL
LIN {X 0,Y 225.74,Z 298.691,A -85,B 0,C 180,E1 -21376.065,E2 -21376.065} C_VEL
LIN {X 0,Y 222.653,Z 293.626,A -85,B 0,C 180,E1 -21377.935,E2 -21377.935} C_VEL
LIN {X 0,Y 219.764,Z 289.134,A -85,B 0,C 180,E1 -21379.887,E2 -21379.887} C_VEL
LIN {X 0,Y 216.756,Z 284.464,A -85,B 0,C 180,E1 -21382.213,E2 -21382.213} C_VEL
LIN {X 0,Y 211.49,Z 277.251,A -85,B 0,C 180,E1 -21387.586,E2 -21387.586} C_VEL
LIN {X 0,Y 207.934,Z 272.906,A -85,B 0,C 180,E1 -21394.402,E2 -21394.402} C_VEL
LIN {X 0,Y 207.46,Z 272.156,A -85,B 0,C 180,E1 -21398.109,E2 -21398.109} C_VEL
LIN {X 0,Y 208.331,Z 273.003,A -85,B 0,C 180,E1 -21402.932,E2 -21402.932} C_VEL
LIN {X 0,Y 212.119,Z 276.782,A -85,B 0,C 180,E1 -21409.271,E2 -21409.271} C_VEL
LIN {X 0,Y 216.613,Z 282.568,A -85,B 0,C 180,E1 -21413.747,E2 -21413.747} C_VEL
LIN {X 0,Y 219.527,Z 286.349,A -85,B 0,C 180,E1 -21415.972,E2 -21415.972} C_VEL
LIN {X 0,Y 220.754,Z 287.855,A -85,B 0,C 180,E1 -21416.821,E2 -21416.821} C_VEL
LIN {X 0,Y 223.872,Z 292.746,A -85,B 0,C 180,E1 -21418.854,E2 -21418.854} C_VEL
LIN {X 0,Y 229.275,Z 301.649,A -85,B 0,C 180,E1 -21421.91,E2 -21421.91} C_VEL
LIN {X 0,Y 233.336,Z 309.549,A -85,B 0,C 180,E1 -21423.972,E2 -21423.972} C_VEL
LIN {X 0,Y 237.473,Z 318.571,A -85,B 0,C 180,E1 -21425.901,E2 -21425.901} C_VEL
LIN {X 0,Y 239.059,Z 322.4,A -85,B 0,C 180,E1 -21426.615,E2 -21426.615} C_VEL
LIN {X 0,Y 235.067,Z 370.865,A -85,B 0,C 180,E1 -21428.329,E2 -21428.329} C_VEL
LIN {X 0,Y 233,Z 384.385,A -85,B 0,C 180,E1 -21429.072,E2 -21429.072} C_VEL
LIN {X 0,Y 230.567,Z 396.619,A -85,B 0,C 180,E1 -21430.082,E2 -21430.082} C_VEL
LIN {X 0,Y 227.659,Z 407.955,A -85,B 0,C 180,E1 -21431.336,E2 -21431.336} C_VEL
LIN {X 0,Y 224.1,Z 419.216,A -85,B 0,C 180,E1 -21432.936,E2 -21432.936} C_VEL
LIN {X 0,Y 220.464,Z 429.209,A -85,B 0,C 180,E1 -21434.762,E2 -21434.762} C_VEL
LIN {X 0,Y 216.535,Z 438.679,A -85,B 0,C 180,E1 -21436.97,E2 -21436.97} C_VEL
LIN {X 0,Y 212.315,Z 447.684,A -85,B 0,C 180,E1 -21439.664,E2 -21439.664} C_VEL
LIN {X 0,Y 208.423,Z 455.338,A -85,B 0,C 180,E1 -21442.644,E2 -21442.644} C_VEL
LIN {X 0,Y 204.878,Z 461.663,A -85,B 0,C 180,E1 -21445.92,E2 -21445.92} C_VEL
LIN {X 0,Y 201.891,Z 466.721,A -85,B 0,C 180,E1 -21449.518,E2 -21449.518} C_VEL
LIN {X 0,Y 200.039,Z 469.66,A -85,B 0,C 180,E1 -21452.529,E2 -21452.529} C_VEL
LIN {X 0,Y 198.591,Z 471.6,A -85,B 0,C 180,E1 -21455.523,E2 -21455.523} C_VEL
LIN {X 0,Y 197.65,Z 472.649,A -85,B 0,C 180,E1 -21458.538,E2 -21458.538} C_VEL
LIN {X 0,Y 196.937,Z 472.695,A -85,B 0,C 180,E1 -21462.669,E2 -21462.669} C_VEL
LIN {X 0,Y 196.753,Z 471.736,A -85,B 0,C 180,E1 -21465.571,E2 -21465.571} C_VEL
LIN {X 0,Y 196.79,Z 469.866,A -85,B 0,C 180,E1 -21468.563,E2 -21468.563} C_VEL
LIN {X 0,Y 197.179,Z 467.009,A -85,B 0,C 180,E1 -21471.615,E2 -21471.615} C_VEL
LIN {X 0,Y 197.795,Z 462.931,A -85,B 0,C 180,E1 -21474.779,E2 -21474.779} C_VEL
LIN {X 0,Y 198.727,Z 457.379,A -85,B 0,C 180,E1 -21478.046,E2 -21478.046} C_VEL
LIN {X 0,Y 200.12,Z 450.013,A -85,B 0,C 180,E1 -21481.364,E2 -21481.364} C_VEL
LIN {X 0,Y 201.869,Z 441.547,A -85,B 0,C 180,E1 -21484.364,E2 -21484.364} C_VEL
LIN {X 0,Y 203.675,Z 432.579,A -85,B 0,C 180,E1 -21486.894,E2 -21486.894} C_VEL
LIN {X 0,Y 205.757,Z 422.084,A -85,B 0,C 180,E1 -21489.249,E2 -21489.249} C_VEL
LIN {X 0,Y 207.779,Z 410.974,A -85,B 0,C 180,E1 -21491.226,E2 -21491.226} C_VEL
LIN {X 0,Y 209.722,Z 398.377,A -85,B 0,C 180,E1 -21492.942,E2 -21492.942} C_VEL
LIN {X 0,Y 211.337,Z 385.078,A -85,B 0,C 180,E1 -21494.291,E2 -21494.291} C_VEL
LIN {X 0,Y 212.596,Z 371.665,A -85,B 0,C 180,E1 -21495.205,E2 -21495.205} C_VEL
LIN {X 0,Y 213.838,Z 349.45,A -85,B 0,C 180,E1 -21496.104,E2 -21496.104} C_VEL
LIN {X 0,Y 215.81,Z 305.066,A -85,B 0,C 180,E1 -21497.768,E2 -21497.768} C_VEL
LIN {X 0,Y 208.719,Z 284.483,A -85,B 0,C 180,E1 -21499.527,E2 -21499.527} C_VEL
LIN {X 0,Y 201.089,Z 265.037,A -85,B 0,C 180,E1 -21501.43,E2 -21501.43} C_VEL
LIN {X 0,Y 200.157,Z 262.691,A -85,B 0,C 180,E1 -21501.803,E2 -21501.803} C_VEL
LIN {X 0,Y 200.068,Z 262.118,A -85,B 0,C 180,E1 -21502.18,E2 -21502.18} C_VEL
LIN {X 0,Y 200.286,Z 262.037,A -85,B 0,C 180,E1 -21507.993,E2 -21507.993} C_VEL
LIN {X 0,Y 200.419,Z 262.012,A -85,B 0,C 180,E1 -21510.003,E2 -21510.003} C_VEL
LIN {X 0,Y 200.287,Z 262.036,A -85,B 0,C 180,E1 -21512.014,E2 -21512.014} C_VEL
LIN {X 0,Y 200.049,Z 262.064,A -85,B 0,C 180,E1 -21518.082,E2 -21518.082} C_VEL
LIN {X 0,Y 199.98,Z 262.058,A -85,B 0,C 180,E1 -21520.353,E2 -21520.353} C_VEL
LIN {X 0,Y 199.739,Z 262.096,A -85,B 0,C 180,E1 -21526.352,E2 -21526.352} C_VEL
LIN {X 0,Y 199.627,Z 262.112,A -85,B 0,C 180,E1 -21530.616,E2 -21530.616} C_VEL
LIN {X 0,Y 199.615,Z 262.116,A -85,B 0,C 180,E1 -21534.996,E2 -21534.996} C_VEL
LIN {X 0,Y 199.619,Z 262.086,A -85,B 0,C 180,E1 -21539.535,E2 -21539.535} C_VEL
LIN {X 0,Y 199.613,Z 262.111,A -85,B 0,C 180,E1 -21542.36,E2 -21542.36} C_VEL
LIN {X 0,Y 199.613,Z 262.117,A -85,B 0,C 180,E1 -21546.769,E2 -21546.769} C_VEL
LIN {X 0,Y 199.641,Z 262.107,A -85,B 0,C 180,E1 -21549.324,E2 -21549.324} C_VEL
LIN {X 0,Y 199.629,Z 262.119,A -85,B 0,C 180,E1 -21552.351,E2 -21552.351} C_VEL
LIN {X 0,Y 199.662,Z 262.107,A -85,B 0,C 180,E1 -21555.275,E2 -21555.275} C_VEL
LIN {X 0,Y 199.665,Z 262.105,A -85,B 0,C 180,E1 -21558.048,E2 -21558.048} C_VEL
LIN {X 0,Y 199.697,Z 262.111,A -85,B 0,C 180,E1 -21560.742,E2 -21560.742} C_VEL
LIN {X 0,Y 199.611,Z 262.108,A -85,B 0,C 180,E1 -21565.732,E2 -21565.732} C_VEL
LIN {X 0,Y 199.676,Z 262.108,A -85,B 0,C 180,E1 -21568.151,E2 -21568.151} C_VEL
LIN {X 0,Y 199.669,Z 262.107,A -85,B 0,C 180,E1 -21572.786,E2 -21572.786} C_VEL
LIN {X 0,Y 199.698,Z 262.105,A -85,B 0,C 180,E1 -21577.24,E2 -21577.24} C_VEL
LIN {X 0,Y 199.739,Z 262.097,A -85,B 0,C 180,E1 -21581.817,E2 -21581.817} C_VEL
LIN {X 0,Y 199.811,Z 262.088,A -85,B 0,C 180,E1 -21585.761,E2 -21585.761} C_VEL
LIN {X 0,Y 200.024,Z 262.066,A -85,B 0,C 180,E1 -21589.896,E2 -21589.896} C_VEL
LIN {X 0,Y 200.008,Z 262.06,A -85,B 0,C 180,E1 -21593.963,E2 -21593.963} C_VEL
LIN {X 0,Y 200.297,Z 262.036,A -85,B 0,C 180,E1 -21598.003,E2 -21598.003} C_VEL
LIN {X 0,Y 200.456,Z 262.009,A -85,B 0,C 180,E1 -21600.013,E2 -21600.013} C_VEL
LIN {X 0,Y 199.996,Z 262.033,A -85,B 0,C 180,E1 -21604.043,E2 -21604.043} C_VEL
LIN {X 0,Y 200.085,Z 262.04,A -85,B 0,C 180,E1 -21608.09,E2 -21608.09} C_VEL
LIN {X 0,Y 199.882,Z 262.087,A -85,B 0,C 180,E1 -21612.192,E2 -21612.192} C_VEL
LIN {X 0,Y 199.777,Z 262.083,A -85,B 0,C 180,E1 -21616.358,E2 -21616.358} C_VEL
LIN {X 0,Y 199.669,Z 262.095,A -85,B 0,C 180,E1 -21620.621,E2 -21620.621} C_VEL
LIN {X 0,Y 199.673,Z 262.112,A -85,B 0,C 180,E1 -21624.997,E2 -21624.997} C_VEL
LIN {X 0,Y 199.635,Z 262.099,A -85,B 0,C 180,E1 -21629.542,E2 -21629.542} C_VEL
LIN {X 0,Y 199.693,Z 262.109,A -85,B 0,C 180,E1 -21632.36,E2 -21632.36} C_VEL
LIN {X 0,Y 199.646,Z 262.1,A -85,B 0,C 180,E1 -21636.772,E2 -21636.772} C_VEL
LIN {X 0,Y 199.624,Z 262.12,A -85,B 0,C 180,E1 -21639.338,E2 -21639.338} C_VEL
LIN {X 0,Y 199.584,Z 262.113,A -85,B 0,C 180,E1 -21642.309,E2 -21642.309} C_VEL
LIN {X 0,Y 199.589,Z 262.123,A -85,B 0,C 180,E1 -21645.227,E2 -21645.227} C_VEL
LIN {X 0,Y 199.59,Z 262.119,A -85,B 0,C 180,E1 -21648.004,E2 -21648.004} C_VEL
LIN {X 0,Y 199.681,Z 262.183,A -85,B 0,C 180,E1 -21651.816,E2 -21651.816} C_VEL
LIN {X 0,Y 200.746,Z 266.976,A -85,B 0,C 180,E1 -21654.331,E2 -21654.331} C_VEL
LIN {X 0,Y 206.003,Z 280.442,A -85,B 0,C 180,E1 -21655.738,E2 -21655.738} C_VEL
LIN {X 0,Y 212.334,Z 297.831,A -85,B 0,C 180,E1 -21657.303,E2 -21657.303} C_VEL
LIN {X 0,Y 212.944,Z 301.609,A -85,B 0,C 180,E1 -21657.541,E2 -21657.541} C_VEL
LIN {X 0,Y 212.738,Z 307.472,A -85,B 0,C 180,E1 -21657.768,E2 -21657.768} C_VEL
LIN {X 0,Y 211.682,Z 313.338,A -85,B 0,C 180,E1 -21657.897,E2 -21657.897} C_VEL
LIN {X 0,Y 208.991,Z 325.282,A -85,B 0,C 180,E1 -21658.11,E2 -21658.11} C_VEL
LIN {X 0,Y 208.478,Z 329.306,A -85,B 0,C 180,E1 -21658.229,E2 -21658.229} C_VEL
LIN {X 0,Y 206.081,Z 374.77,A -85,B 0,C 180,E1 -21660.008,E2 -21660.008} C_VEL
LIN {X 0,Y 204.853,Z 388.75,A -85,B 0,C 180,E1 -21660.941,E2 -21660.941} C_VEL
LIN {X 0,Y 203.267,Z 401.405,A -85,B 0,C 180,E1 -21662.172,E2 -21662.172} C_VEL
LIN {X 0,Y 201.08,Z 413.841,A -85,B 0,C 180,E1 -21663.812,E2 -21663.812} C_VEL
LIN {X 0,Y 199.028,Z 425.111,A -85,B 0,C 180,E1 -21665.761,E2 -21665.761} C_VEL
LIN {X 0,Y 197.2,Z 434.696,A -85,B 0,C 180,E1 -21667.854,E2 -21667.854} C_VEL
LIN {X 0,Y 195.174,Z 444.514,A -85,B 0,C 180,E1 -21670.541,E2 -21670.541} C_VEL
LIN {X 0,Y 193.277,Z 453.488,A -85,B 0,C 180,E1 -21673.628,E2 -21673.628} C_VEL
LIN {X 0,Y 191.829,Z 460.62,A -85,B 0,C 180,E1 -21676.76,E2 -21676.76} C_VEL
LIN {X 0,Y 190.786,Z 467.131,A -85,B 0,C 180,E1 -21680.455,E2 -21680.455} C_VEL
LIN {X 0,Y 190.312,Z 471.368,A -85,B 0,C 180,E1 -21683.636,E2 -21683.636} C_VEL
LIN {X 0,Y 190.128,Z 474.287,A -85,B 0,C 180,E1 -21686.579,E2 -21686.579} C_VEL
LIN {X 0,Y 190.188,Z 476.596,A -85,B 0,C 180,E1 -21689.996,E2 -21689.996} C_VEL
LIN {X 0,Y 190.093,Z 477.754,A -85,B 0,C 180,E1 -21693.243,E2 -21693.243} C_VEL
LIN {X 0,Y 190.329,Z 477.98,A -85,B 0,C 180,E1 -21696.356,E2 -21696.356} C_VEL
LIN {X 0,Y 191.267,Z 476.921,A -85,B 0,C 180,E1 -21700.583,E2 -21700.583} C_VEL
LIN {X 0,Y 192.04,Z 475.808,A -85,B 0,C 180,E1 -21702.68,E2 -21702.68} C_VEL
LIN {X 0,Y 194.208,Z 472.299,A -85,B 0,C 180,E1 -21706.824,E2 -21706.824} C_VEL
LIN {X 0,Y 196.675,Z 468.521,A -85,B 0,C 180,E1 -21709.841,E2 -21709.841} C_VEL
LIN {X 0,Y 199.683,Z 463.665,A -85,B 0,C 180,E1 -21712.773,E2 -21712.773} C_VEL
LIN {X 0,Y 202.844,Z 457.965,A -85,B 0,C 180,E1 -21715.489,E2 -21715.489} C_VEL
LIN {X 0,Y 206.854,Z 450.165,A -85,B 0,C 180,E1 -21718.398,E2 -21718.398} C_VEL
LIN {X 0,Y 210.521,Z 442.587,A -85,B 0,C 180,E1 -21720.6,E2 -21720.6} C_VEL
LIN {X 0,Y 214.562,Z 433.436,A -85,B 0,C 180,E1 -21722.71,E2 -21722.71} C_VEL
LIN {X 0,Y 218.837,Z 422.16,A -85,B 0,C 180,E1 -21724.749,E2 -21724.749} C_VEL
LIN {X 0,Y 222.556,Z 410.96,A -85,B 0,C 180,E1 -21726.301,E2 -21726.301} C_VEL
LIN {X 0,Y 225.928,Z 398.33,A -85,B 0,C 180,E1 -21727.62,E2 -21727.62} C_VEL
LIN {X 0,Y 228.79,Z 384.881,A -85,B 0,C 180,E1 -21728.603,E2 -21728.603} C_VEL
LIN {X 0,Y 230.732,Z 371.059,A -85,B 0,C 180,E1 -21729.269,E2 -21729.269} C_VEL
LIN {X 0,Y 234.269,Z 328.921,A -85,B 0,C 180,E1 -21730.752,E2 -21730.752} C_VEL
LIN {X 0,Y 230.369,Z 319.151,A -85,B 0,C 180,E1 -21732.723,E2 -21732.723} C_VEL
LIN {X 0,Y 226.985,Z 312.04,A -85,B 0,C 180,E1 -21734.515,E2 -21734.515} C_VEL
LIN {X 0,Y 223.012,Z 304.517,A -85,B 0,C 180,E1 -21736.842,E2 -21736.842} C_VEL
LIN {X 0,Y 220.11,Z 299.606,A -85,B 0,C 180,E1 -21738.693,E2 -21738.693} C_VEL
LIN {X 0,Y 217.57,Z 295.401,A -85,B 0,C 180,E1 -21740.553,E2 -21740.553} C_VEL
LIN {X 0,Y 214.287,Z 290.239,A -85,B 0,C 180,E1 -21743.294,E2 -21743.294} C_VEL
LIN {X 0,Y 210.02,Z 284.009,A -85,B 0,C 180,E1 -21748.025,E2 -21748.025} C_VEL
LIN {X 0,Y 206.769,Z 279.801,A -85,B 0,C 180,E1 -21754.728,E2 -21754.728} C_VEL
LIN {X 0,Y 206.37,Z 279.164,A -85,B 0,C 180,E1 -21757.988,E2 -21757.988} C_VEL
LIN {X 0,Y 207.276,Z 280.08,A -85,B 0,C 180,E1 -21763.078,E2 -21763.078} C_VEL
LIN {X 0,Y 210.699,Z 283.689,A -85,B 0,C 180,E1 -21768.935,E2 -21768.935} C_VEL
LIN {X 0,Y 214.747,Z 289.084,A -85,B 0,C 180,E1 -21773.176,E2 -21773.176} C_VEL
LIN {X 0,Y 217.614,Z 292.937,A -85,B 0,C 180,E1 -21775.494,E2 -21775.494} C_VEL
LIN {X 0,Y 218.658,Z 294.348,A -85,B 0,C 180,E1 -21776.255,E2 -21776.255} C_VEL
LIN {X 0,Y 221.335,Z 298.772,A -85,B 0,C 180,E1 -21778.131,E2 -21778.131} C_VEL
LIN {X 0,Y 226.343,Z 307.45,A -85,B 0,C 180,E1 -21781.156,E2 -21781.156} C_VEL
LIN {X 0,Y 229.617,Z 313.958,A -85,B 0,C 180,E1 -21782.909,E2 -21782.909} C_VEL
LIN {X 0,Y 233.716,Z 323.277,A -85,B 0,C 180,E1 -21784.992,E2 -21784.992} C_VEL
LIN {X 0,Y 234.458,Z 325.073,A -85,B 0,C 180,E1 -21785.344,E2 -21785.344} C_VEL
LIN {X 0,Y 230.509,Z 371.086,A -85,B 0,C 180,E1 -21786.993,E2 -21786.993} C_VEL
LIN {X 0,Y 228.432,Z 384.308,A -85,B 0,C 180,E1 -21787.726,E2 -21787.726} C_VEL
LIN {X 0,Y 225.873,Z 396.397,A -85,B 0,C 180,E1 -21788.712,E2 -21788.712} C_VEL
LIN {X 0,Y 222.848,Z 407.691,A -85,B 0,C 180,E1 -21789.966,E2 -21789.966} C_VEL
LIN {X 0,Y 219.188,Z 418.773,A -85,B 0,C 180,E1 -21791.547,E2 -21791.547} C_VEL
LIN {X 0,Y 215.248,Z 429.101,A -85,B 0,C 180,E1 -21793.439,E2 -21793.439} C_VEL
LIN {X 0,Y 211.465,Z 437.887,A -85,B 0,C 180,E1 -21795.477,E2 -21795.477} C_VEL
LIN {X 0,Y 207.051,Z 446.857,A -85,B 0,C 180,E1 -21798.132,E2 -21798.132} C_VEL
LIN {X 0,Y 203.135,Z 454.145,A -85,B 0,C 180,E1 -21800.922,E2 -21800.922} C_VEL
LIN {X 0,Y 199.714,Z 459.994,A -85,B 0,C 180,E1 -21803.812,E2 -21803.812} C_VEL
LIN {X 0,Y 196.828,Z 464.626,A -85,B 0,C 180,E1 -21806.8,E2 -21806.8} C_VEL
LIN {X 0,Y 194.094,Z 468.718,A -85,B 0,C 180,E1 -21810.441,E2 -21810.441} C_VEL
LIN {X 0,Y 192.562,Z 470.82,A -85,B 0,C 180,E1 -21813.174,E2 -21813.174} C_VEL
LIN {X 0,Y 191.255,Z 472.245,A -85,B 0,C 180,E1 -21816.065,E2 -21816.065} C_VEL
LIN {X 0,Y 190.394,Z 472.936,A -85,B 0,C 180,E1 -21819.186,E2 -21819.186} C_VEL
LIN {X 0,Y 189.892,Z 472.786,A -85,B 0,C 180,E1 -21822.257,E2 -21822.257} C_VEL
LIN {X 0,Y 189.675,Z 471.824,A -85,B 0,C 180,E1 -21825.257,E2 -21825.257} C_VEL
LIN {X 0,Y 189.67,Z 470.074,A -85,B 0,C 180,E1 -21828.172,E2 -21828.172} C_VEL
LIN {X 0,Y 189.971,Z 467.576,A -85,B 0,C 180,E1 -21831.035,E2 -21831.035} C_VEL
LIN {X 0,Y 190.556,Z 463.814,A -85,B 0,C 180,E1 -21834.203,E2 -21834.203} C_VEL
LIN {X 0,Y 191.443,Z 458.519,A -85,B 0,C 180,E1 -21837.57,E2 -21837.57} C_VEL
LIN {X 0,Y 192.785,Z 451.537,A -85,B 0,C 180,E1 -21841,E2 -21841} C_VEL
LIN {X 0,Y 194.235,Z 444.614,A -85,B 0,C 180,E1 -21843.694,E2 -21843.694} C_VEL
LIN {X 0,Y 196.099,Z 435.628,A -85,B 0,C 180,E1 -21846.507,E2 -21846.507} C_VEL
LIN {X 0,Y 198.197,Z 425.634,A -85,B 0,C 180,E1 -21849.006,E2 -21849.006} C_VEL
LIN {X 0,Y 200.366,Z 414.403,A -85,B 0,C 180,E1 -21851.218,E2 -21851.218} C_VEL
LIN {X 0,Y 202.428,Z 402.054,A -85,B 0,C 180,E1 -21853.1,E2 -21853.1} C_VEL
LIN {X 0,Y 204.149,Z 389.871,A -85,B 0,C 180,E1 -21854.5,E2 -21854.5} C_VEL
LIN {X 0,Y 205.566,Z 376.129,A -85,B 0,C 180,E1 -21855.621,E2 -21855.621} C_VEL
LIN {X 0,Y 206.586,Z 362.549,A -85,B 0,C 180,E1 -21856.314,E2 -21856.314} C_VEL
LIN {X 0,Y 209.266,Z 306.553,A -85,B 0,C 180,E1 -21858.475,E2 -21858.475} C_VEL
LIN {X 0,Y 202.066,Z 285.685,A -85,B 0,C 180,E1 -21860.336,E2 -21860.336} C_VEL
LIN {X 0,Y 195.231,Z 268.382,A -85,B 0,C 180,E1 -21862.115,E2 -21862.115} C_VEL
LIN {X 0,Y 193.157,Z 263.816,A -85,B 0,C 180,E1 -21862.753,E2 -21862.753} C_VEL
LIN {X 0,Y 192.96,Z 263.002,A -85,B 0,C 180,E1 -21863.206,E2 -21863.206} C_VEL
LIN {X 0,Y 193.225,Z 262.917,A -85,B 0,C 180,E1 -21867.919,E2 -21867.919} C_VEL
LIN {X 0,Y 193.384,Z 262.888,A -85,B 0,C 180,E1 -21870.004,E2 -21870.004} C_VEL
LIN {X 0,Y 192.93,Z 262.94,A -85,B 0,C 180,E1 -21874.182,E2 -21874.182} C_VEL
LIN {X 0,Y 193.001,Z 262.941,A -85,B 0,C 180,E1 -21878.379,E2 -21878.379} C_VEL
LIN {X 0,Y 192.743,Z 262.972,A -85,B 0,C 180,E1 -21882.641,E2 -21882.641} C_VEL
LIN {X 0,Y 192.697,Z 262.965,A -85,B 0,C 180,E1 -21886.968,E2 -21886.968} C_VEL
LIN {X 0,Y 192.563,Z 262.993,A -85,B 0,C 180,E1 -21891.409,E2 -21891.409} C_VEL
LIN {X 0,Y 192.597,Z 262.991,A -85,B 0,C 180,E1 -21894.222,E2 -21894.222} C_VEL
LIN {X 0,Y 192.598,Z 262.957,A -85,B 0,C 180,E1 -21898.899,E2 -21898.899} C_VEL
LIN {X 0,Y 192.556,Z 262.995,A -85,B 0,C 180,E1 -21903.198,E2 -21903.198} C_VEL
LIN {X 0,Y 192.562,Z 262.989,A -85,B 0,C 180,E1 -21908.353,E2 -21908.353} C_VEL
LIN {X 0,Y 192.579,Z 262.995,A -85,B 0,C 180,E1 -21913.148,E2 -21913.148} C_VEL
LIN {X 0,Y 192.598,Z 262.983,A -85,B 0,C 180,E1 -21916.875,E2 -21916.875} C_VEL
LIN {X 0,Y 192.602,Z 262.991,A -85,B 0,C 180,E1 -21921.681,E2 -21921.681} C_VEL
LIN {X 0,Y 192.577,Z 262.987,A -85,B 0,C 180,E1 -21926.829,E2 -21926.829} C_VEL
LIN {X 0,Y 192.644,Z 262.984,A -85,B 0,C 180,E1 -21931.706,E2 -21931.706} C_VEL
LIN {X 0,Y 192.672,Z 262.977,A -85,B 0,C 180,E1 -21936.361,E2 -21936.361} C_VEL
LIN {X 0,Y 192.688,Z 262.977,A -85,B 0,C 180,E1 -21941.507,E2 -21941.507} C_VEL
LIN {X 0,Y 192.735,Z 262.965,A -85,B 0,C 180,E1 -21945.227,E2 -21945.227} C_VEL
LIN {X 0,Y 192.946,Z 262.95,A -85,B 0,C 180,E1 -21949.582,E2 -21949.582} C_VEL
LIN {X 0,Y 192.972,Z 262.935,A -85,B 0,C 180,E1 -21953.742,E2 -21953.742} C_VEL
LIN {X 0,Y 193.241,Z 262.915,A -85,B 0,C 180,E1 -21957.93,E2 -21957.93} C_VEL
LIN {X 0,Y 193.422,Z 262.884,A -85,B 0,C 180,E1 -21960.014,E2 -21960.014} C_VEL
